// LS Electric XG5000 project: JG FRT C_MBR MAIN WELD
// PLC NewPLC
// module base 0 slot 0: 입력 모듈:XGI-D24A/B (DC 24V 입력, 32점 (전류소스 싱크공용/ 전류소스 입력))
// module base 0 slot 1: 출력 모듈:XGQ-TR4A/B (트랜지스터 출력, 32점 (0.1A용, 싱크출력/소스출력))
// module base 0 slot 2: 출력 모듈:XGQ-TR4A/B (트랜지스터 출력, 32점 (0.1A용, 싱크출력/소스출력))
// module base 0 slot 3: Rnet:XGL-RMEA/B (Rnet 통신 모듈, Rnet Master)
// module base 0 slot 4: Rnet:XGL-RMEA/B (Rnet 통신 모듈, Rnet Master)
// module base 0 slot 5: Rnet:XGL-RMEA/B (Rnet 통신 모듈, Rnet Master)
// module base 0 slot 6: Dnet:XGL-DMEA/B (Dnet 통신 모듈, DeviceNet Master)
// module base 0 slot 7: Dnet:XGL-DMEA/B (Dnet 통신 모듈, DeviceNet Master)
// module base 0 slot 8: FEnet:XGL-EFMT(B) (Fast Ethernet 통신 모듈, 전기 Master)
// module base 0 slot 9: FEnet:XGL-EFMT(B) (Fast Ethernet 통신 모듈, 전기 Master)

PROGRAM Main (task: 스캔 프로그램)

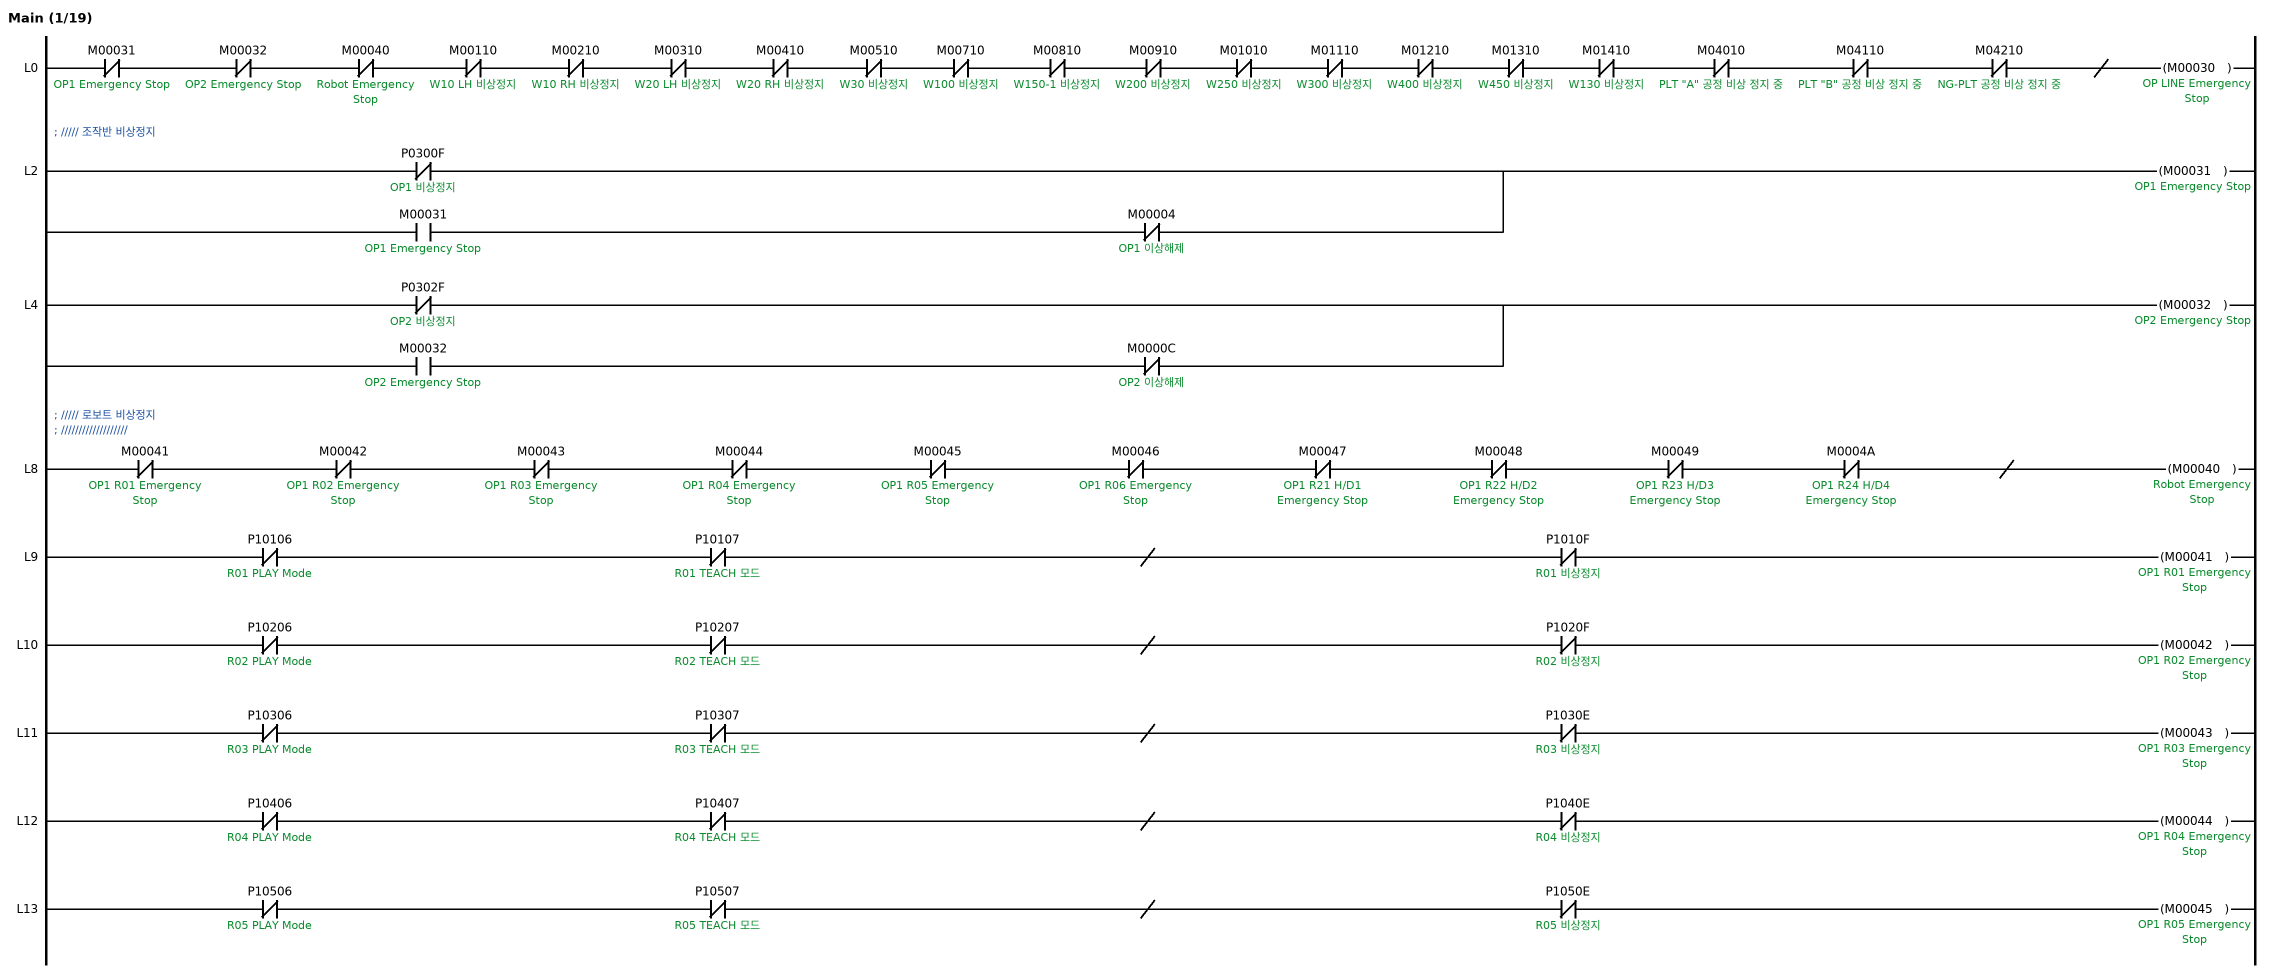
; L0
LOAD NOT  M00031	// OP1 Emergency Stop
AND NOT   M00032	// OP2 Emergency Stop
AND NOT   M00040	// Robot Emergency Stop
AND NOT   M00110	// W10 LH 비상정지
AND NOT   M00210	// W10 RH 비상정지
AND NOT   M00310	// W20 LH 비상정지
AND NOT   M00410	// W20 RH 비상정지
AND NOT   M00510	// W30 비상정지
AND NOT   M00710	// W100 비상정지
AND NOT   M00810	// W150-1 비상정지
AND NOT   M00910	// W200 비상정지
AND NOT   M01010	// W250 비상정지
AND NOT   M01110	// W300 비상정지
AND NOT   M01210	// W400 비상정지
AND NOT   M01310	// W450 비상정지
AND NOT   M01410	// W130 비상정지
AND NOT   M04010	// PLT "A" 공정 비상 정지 중
AND NOT   M04110	// PLT "B" 공정 비상 정지 중
AND NOT   M04210	// NG-PLT 공정 비상 정지 중
NOT
OUT       M00030	// OP LINE Emergency Stop
// ///// 조작반 비상정지
; L2
LOAD NOT  P0300F	// OP1 비상정지
LOAD      M00031	// OP1 Emergency Stop
AND NOT   M00004	// OP1 이상해제
OR LOAD
OUT       M00031	// OP1 Emergency Stop
; L4
LOAD NOT  P0302F	// OP2 비상정지
LOAD      M00032	// OP2 Emergency Stop
AND NOT   M0000C	// OP2 이상해제
OR LOAD
OUT       M00032	// OP2 Emergency Stop
// ///// 로보트 비상정지
// ///////////////////
; L8
LOAD NOT  M00041	// OP1 R01 Emergency Stop
AND NOT   M00042	// OP1 R02 Emergency Stop
AND NOT   M00043	// OP1 R03 Emergency Stop
AND NOT   M00044	// OP1 R04 Emergency Stop
AND NOT   M00045	// OP1 R05 Emergency Stop
AND NOT   M00046	// OP1 R06 Emergency Stop
AND NOT   M00047	// OP1 R21 H/D1 Emergency Stop
AND NOT   M00048	// OP1 R22 H/D2 Emergency Stop
AND NOT   M00049	// OP1 R23 H/D3 Emergency Stop
AND NOT   M0004A	// OP1 R24 H/D4 Emergency Stop
NOT
OUT       M00040	// Robot Emergency Stop
; L9
LOAD NOT  P10106	// R01 PLAY Mode
AND NOT   P10107	// R01 TEACH 모드
NOT
AND NOT   P1010F	// R01 비상정지
OUT       M00041	// OP1 R01 Emergency Stop
; L10
LOAD NOT  P10206	// R02 PLAY Mode
AND NOT   P10207	// R02 TEACH 모드
NOT
AND NOT   P1020F	// R02 비상정지
OUT       M00042	// OP1 R02 Emergency Stop
; L11
LOAD NOT  P10306	// R03 PLAY Mode
AND NOT   P10307	// R03 TEACH 모드
NOT
AND NOT   P1030E	// R03 비상정지
OUT       M00043	// OP1 R03 Emergency Stop
; L12
LOAD NOT  P10406	// R04 PLAY Mode
AND NOT   P10407	// R04 TEACH 모드
NOT
AND NOT   P1040E	// R04 비상정지
OUT       M00044	// OP1 R04 Emergency Stop
; L13
LOAD NOT  P10506	// R05 PLAY Mode
AND NOT   P10507	// R05 TEACH 모드
NOT
AND NOT   P1050E	// R05 비상정지
OUT       M00045	// OP1 R05 Emergency Stop

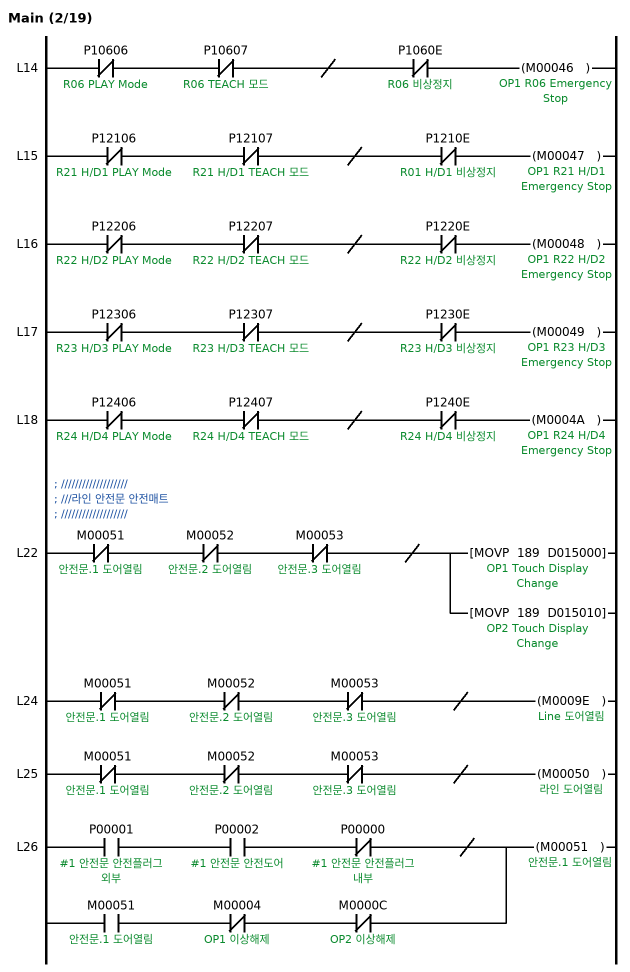
; L14
LOAD NOT  P10606	// R06 PLAY Mode
AND NOT   P10607	// R06 TEACH 모드
NOT
AND NOT   P1060E	// R06 비상정지
OUT       M00046	// OP1 R06 Emergency Stop
; L15
LOAD NOT  P12106	// R21 H/D1 PLAY Mode
AND NOT   P12107	// R21 H/D1 TEACH 모드
NOT
AND NOT   P1210E	// R01 H/D1 비상정지
OUT       M00047	// OP1 R21 H/D1 Emergency Stop
; L16
LOAD NOT  P12206	// R22 H/D2 PLAY Mode
AND NOT   P12207	// R22 H/D2 TEACH 모드
NOT
AND NOT   P1220E	// R22 H/D2 비상정지
OUT       M00048	// OP1 R22 H/D2 Emergency Stop
; L17
LOAD NOT  P12306	// R23 H/D3 PLAY Mode
AND NOT   P12307	// R23 H/D3 TEACH 모드
NOT
AND NOT   P1230E	// R23 H/D3 비상정지
OUT       M00049	// OP1 R23 H/D3 Emergency Stop
; L18
LOAD NOT  P12406	// R24 H/D4 PLAY Mode
AND NOT   P12407	// R24 H/D4 TEACH 모드
NOT
AND NOT   P1240E	// R24 H/D4 비상정지
OUT       M0004A	// OP1 R24 H/D4 Emergency Stop
// ///////////////////
// ///라인 안전문 안전매트
// ///////////////////
; L22
LOAD NOT  M00051	// 안전문.1 도어열림
AND NOT   M00052	// 안전문.2 도어열림
AND NOT   M00053	// 안전문.3 도어열림
NOT
MOVP      189 D015000	// OP1 Touch Display Change
MOVP      189 D015010	// OP2 Touch Display Change
; L24
LOAD NOT  M00051	// 안전문.1 도어열림
AND NOT   M00052	// 안전문.2 도어열림
AND NOT   M00053	// 안전문.3 도어열림
NOT
OUT       M0009E	// Line 도어열림
; L25
LOAD NOT  M00051	// 안전문.1 도어열림
AND NOT   M00052	// 안전문.2 도어열림
AND NOT   M00053	// 안전문.3 도어열림
NOT
OUT       M00050	// 라인 도어열림
; L26
LOAD      P00001	// #1 안전문 안전플러그 외부
AND       P00002	// #1 안전문 안전도어
AND NOT   P00000	// #1 안전문 안전플러그 내부
NOT
LOAD      M00051	// 안전문.1 도어열림
AND NOT   M00004	// OP1 이상해제
AND NOT   M0000C	// OP2 이상해제
OR LOAD
OUT       M00051	// 안전문.1 도어열림

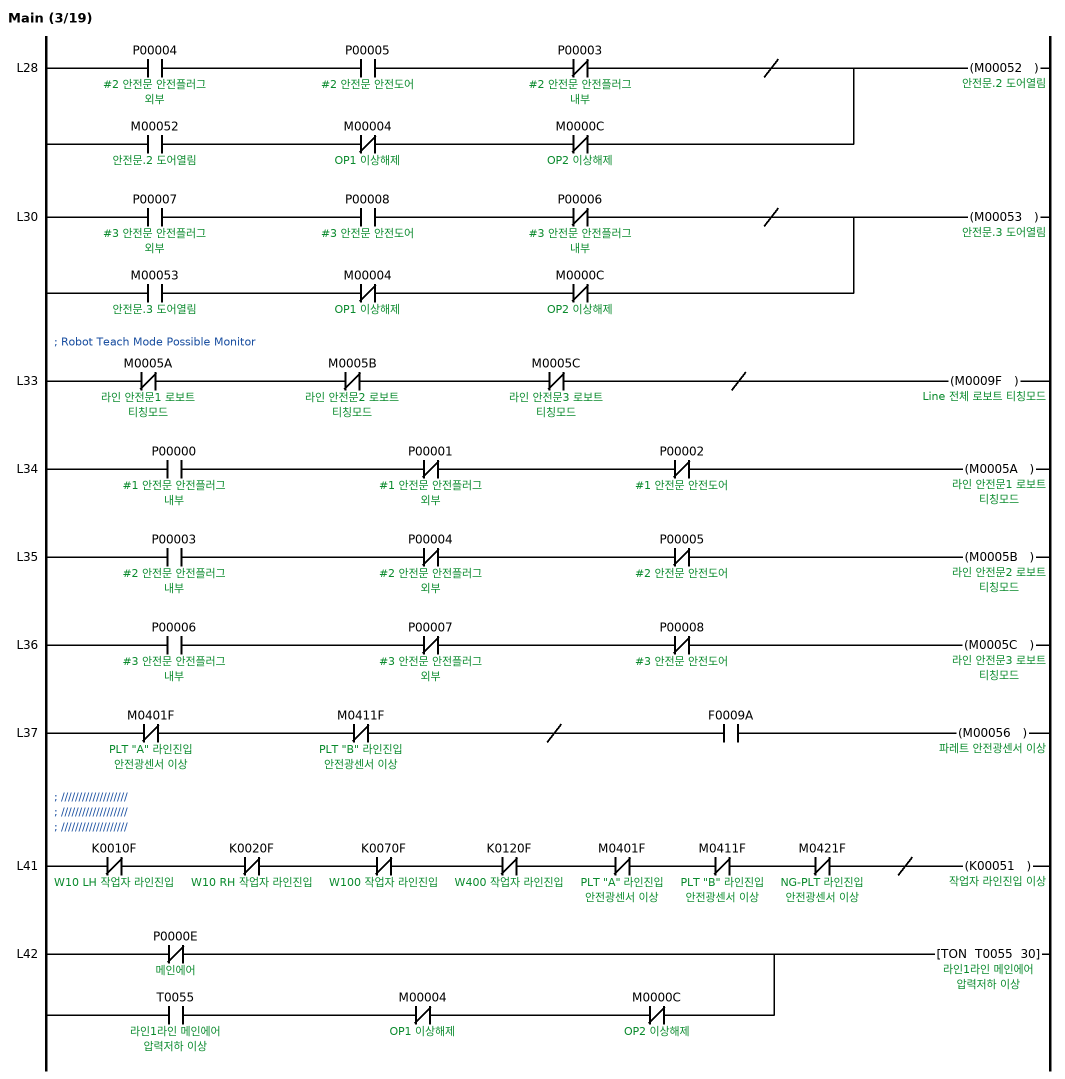
; L28
LOAD      P00004	// #2 안전문 안전플러그 외부
AND       P00005	// #2 안전문 안전도어
AND NOT   P00003	// #2 안전문 안전플러그 내부
NOT
LOAD      M00052	// 안전문.2 도어열림
AND NOT   M00004	// OP1 이상해제
AND NOT   M0000C	// OP2 이상해제
OR LOAD
OUT       M00052	// 안전문.2 도어열림
; L30
LOAD      P00007	// #3 안전문 안전플러그 외부
AND       P00008	// #3 안전문 안전도어
AND NOT   P00006	// #3 안전문 안전플러그 내부
NOT
LOAD      M00053	// 안전문.3 도어열림
AND NOT   M00004	// OP1 이상해제
AND NOT   M0000C	// OP2 이상해제
OR LOAD
OUT       M00053	// 안전문.3 도어열림
// Robot Teach Mode Possible Monitor
; L33
LOAD NOT  M0005A	// 라인 안전문1 로보트 티칭모드
AND NOT   M0005B	// 라인 안전문2 로보트 티칭모드
AND NOT   M0005C	// 라인 안전문3 로보트 티칭모드
NOT
OUT       M0009F	// Line 전체 로보트 티칭모드
; L34
LOAD      P00000	// #1 안전문 안전플러그 내부
AND NOT   P00001	// #1 안전문 안전플러그 외부
AND NOT   P00002	// #1 안전문 안전도어
OUT       M0005A	// 라인 안전문1 로보트 티칭모드
; L35
LOAD      P00003	// #2 안전문 안전플러그 내부
AND NOT   P00004	// #2 안전문 안전플러그 외부
AND NOT   P00005	// #2 안전문 안전도어
OUT       M0005B	// 라인 안전문2 로보트 티칭모드
; L36
LOAD      P00006	// #3 안전문 안전플러그 내부
AND NOT   P00007	// #3 안전문 안전플러그 외부
AND NOT   P00008	// #3 안전문 안전도어
OUT       M0005C	// 라인 안전문3 로보트 티칭모드
; L37
LOAD NOT  M0401F	// PLT "A" 라인진입 안전광센서 이상
AND NOT   M0411F	// PLT "B" 라인진입 안전광센서 이상
NOT
AND       F0009A
OUT       M00056	// 파레트 안전광센서 이상
// ///////////////////
// ///////////////////
// ///////////////////
; L41
LOAD NOT  K0010F	// W10 LH 작업자 라인진입
AND NOT   K0020F	// W10 RH 작업자 라인진입
AND NOT   K0070F	// W100 작업자 라인진입
AND NOT   K0120F	// W400 작업자 라인진입
AND NOT   M0401F	// PLT "A" 라인진입 안전광센서 이상
AND NOT   M0411F	// PLT "B" 라인진입 안전광센서 이상
AND NOT   M0421F	// NG-PLT 라인진입 안전광센서 이상
NOT
OUT       K00051	//  작업자 라인진입 이상
; L42
LOAD NOT  P0000E	// 메인에어
LOAD      T0055	// 라인1라인 메인에어 압력저하 이상
AND NOT   M00004	// OP1 이상해제
AND NOT   M0000C	// OP2 이상해제
OR LOAD
TON       T0055 30	// 라인1라인 메인에어 압력저하 이상

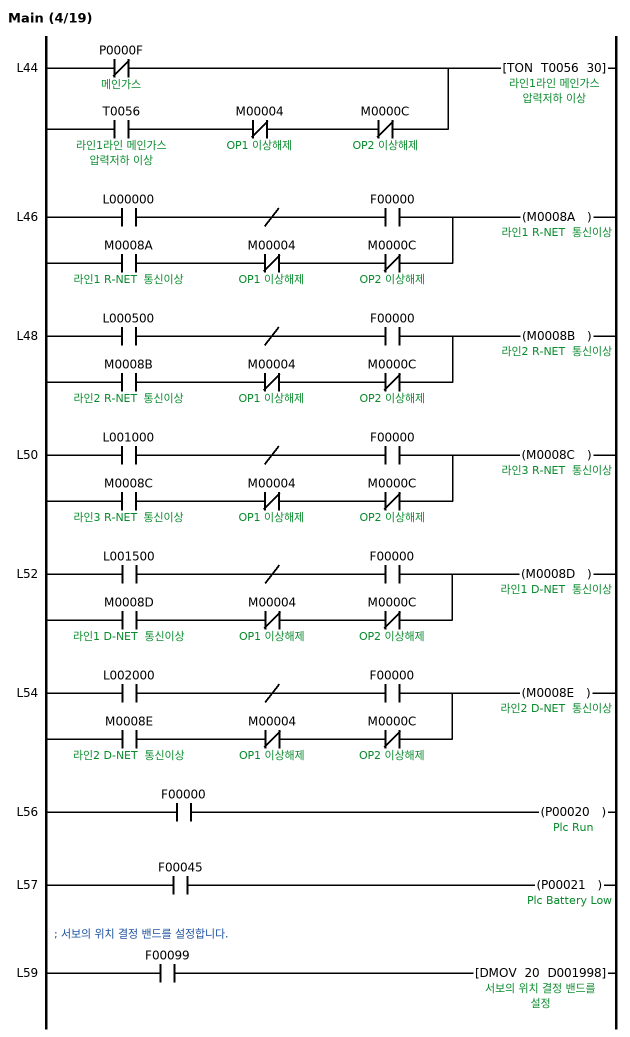
; L44
LOAD NOT  P0000F	// 메인가스
LOAD      T0056	// 라인1라인 메인가스 압력저하 이상
AND NOT   M00004	// OP1 이상해제
AND NOT   M0000C	// OP2 이상해제
OR LOAD
TON       T0056 30	// 라인1라인 메인가스 압력저하 이상
; L46
LOAD      L000000
NOT
AND       F00000
LOAD      M0008A	// 라인1 R-NET  통신이상
AND NOT   M00004	// OP1 이상해제
AND NOT   M0000C	// OP2 이상해제
OR LOAD
OUT       M0008A	// 라인1 R-NET  통신이상
; L48
LOAD      L000500
NOT
AND       F00000
LOAD      M0008B	// 라인2 R-NET  통신이상
AND NOT   M00004	// OP1 이상해제
AND NOT   M0000C	// OP2 이상해제
OR LOAD
OUT       M0008B	// 라인2 R-NET  통신이상
; L50
LOAD      L001000
NOT
AND       F00000
LOAD      M0008C	// 라인3 R-NET  통신이상
AND NOT   M00004	// OP1 이상해제
AND NOT   M0000C	// OP2 이상해제
OR LOAD
OUT       M0008C	// 라인3 R-NET  통신이상
; L52
LOAD      L001500
NOT
AND       F00000
LOAD      M0008D	// 라인1 D-NET  통신이상
AND NOT   M00004	// OP1 이상해제
AND NOT   M0000C	// OP2 이상해제
OR LOAD
OUT       M0008D	// 라인1 D-NET  통신이상
; L54
LOAD      L002000
NOT
AND       F00000
LOAD      M0008E	// 라인2 D-NET  통신이상
AND NOT   M00004	// OP1 이상해제
AND NOT   M0000C	// OP2 이상해제
OR LOAD
OUT       M0008E	// 라인2 D-NET  통신이상
; L56
LOAD      F00000
OUT       P00020	// Plc Run
; L57
LOAD      F00045
OUT       P00021	// Plc Battery Low
// 서보의 위치 결정 밴드를 설정합니다.
; L59
LOAD      F00099
DMOV      20 D001998	// 서보의 위치 결정 밴드를 설정

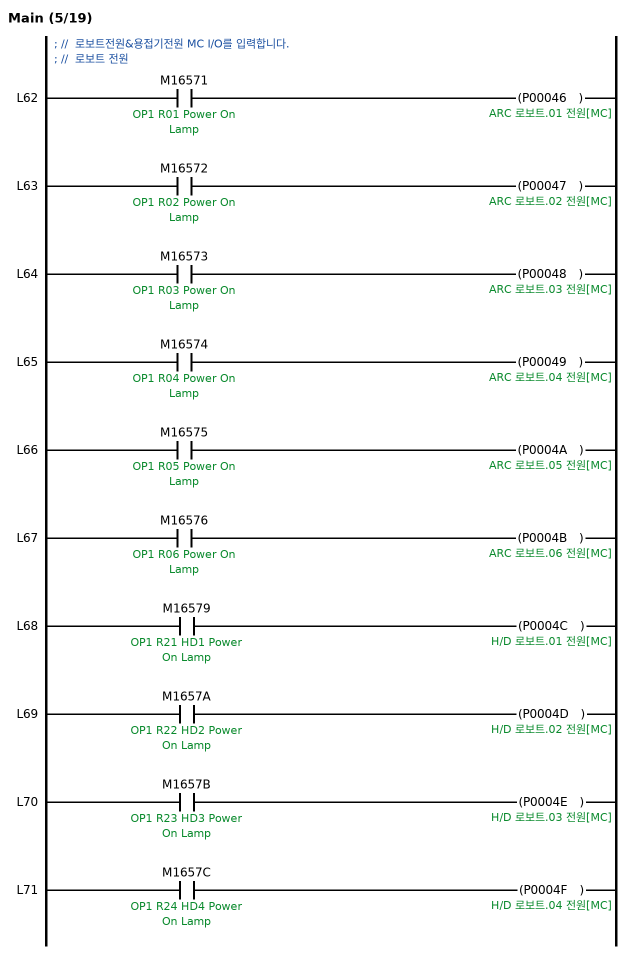
//   //  로보트전원&용접기전원 MC I/O를 입력합니다.
//   //  로보트 전원
; L62
LOAD      M16571	// OP1 R01 Power On Lamp
OUT       P00046	// ARC 로보트.01 전원[MC]
; L63
LOAD      M16572	// OP1 R02 Power On Lamp
OUT       P00047	// ARC 로보트.02 전원[MC]
; L64
LOAD      M16573	// OP1 R03 Power On Lamp
OUT       P00048	// ARC 로보트.03 전원[MC]
; L65
LOAD      M16574	// OP1 R04 Power On Lamp
OUT       P00049	// ARC 로보트.04 전원[MC]
; L66
LOAD      M16575	// OP1 R05 Power On Lamp
OUT       P0004A	// ARC 로보트.05 전원[MC]
; L67
LOAD      M16576	// OP1 R06 Power On Lamp
OUT       P0004B	// ARC 로보트.06 전원[MC]
; L68
LOAD      M16579	// OP1 R21 HD1 Power On Lamp
OUT       P0004C	// H/D 로보트.01 전원[MC]
; L69
LOAD      M1657A	// OP1 R22 HD2 Power On Lamp
OUT       P0004D	// H/D 로보트.02 전원[MC]
; L70
LOAD      M1657B	// OP1 R23 HD3 Power On Lamp
OUT       P0004E	// H/D 로보트.03 전원[MC]
; L71
LOAD      M1657C	// OP1 R24 HD4 Power On Lamp
OUT       P0004F	// H/D 로보트.04 전원[MC]

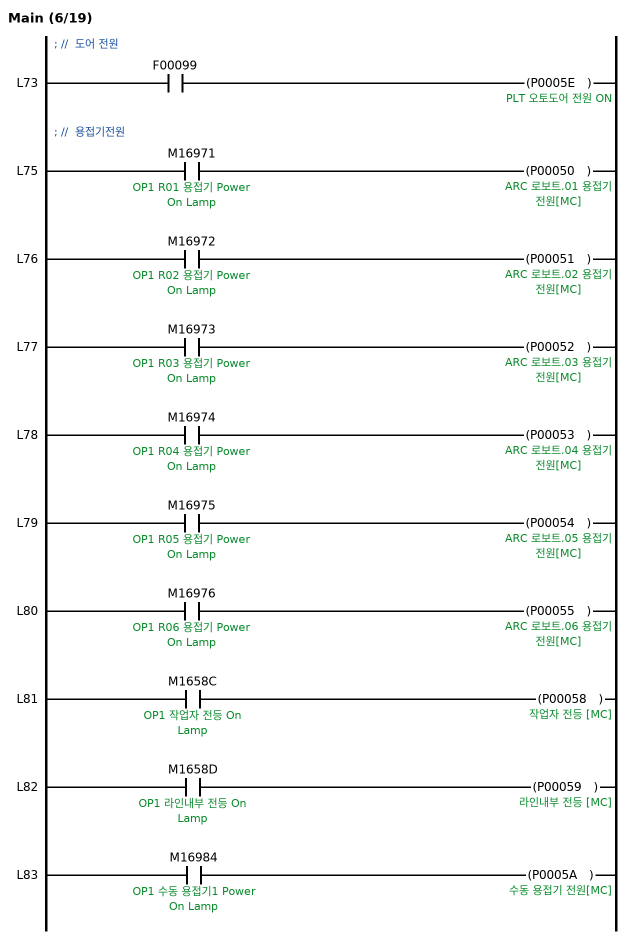
//   //  도어 전원
; L73
LOAD      F00099
OUT       P0005E	// PLT 오토도어 전원 ON
//   //  용접기전원
; L75
LOAD      M16971	// OP1 R01 용접기 Power On Lamp
OUT       P00050	// ARC 로보트.01 용접기 전원[MC]
; L76
LOAD      M16972	// OP1 R02 용접기 Power On Lamp
OUT       P00051	// ARC 로보트.02 용접기 전원[MC]
; L77
LOAD      M16973	// OP1 R03 용접기 Power On Lamp
OUT       P00052	// ARC 로보트.03 용접기 전원[MC]
; L78
LOAD      M16974	// OP1 R04 용접기 Power On Lamp
OUT       P00053	// ARC 로보트.04 용접기 전원[MC]
; L79
LOAD      M16975	// OP1 R05 용접기 Power On Lamp
OUT       P00054	// ARC 로보트.05 용접기 전원[MC]
; L80
LOAD      M16976	// OP1 R06 용접기 Power On Lamp
OUT       P00055	// ARC 로보트.06 용접기 전원[MC]
; L81
LOAD      M1658C	// OP1 작업자 전등 On Lamp
OUT       P00058	// 작업자 전등 [MC]
; L82
LOAD      M1658D	// OP1 라인내부 전등 On Lamp
OUT       P00059	// 라인내부 전등 [MC]
; L83
LOAD      M16984	// OP1 수동 용접기1 Power On Lamp
OUT       P0005A	// 수동 용접기 전원[MC]

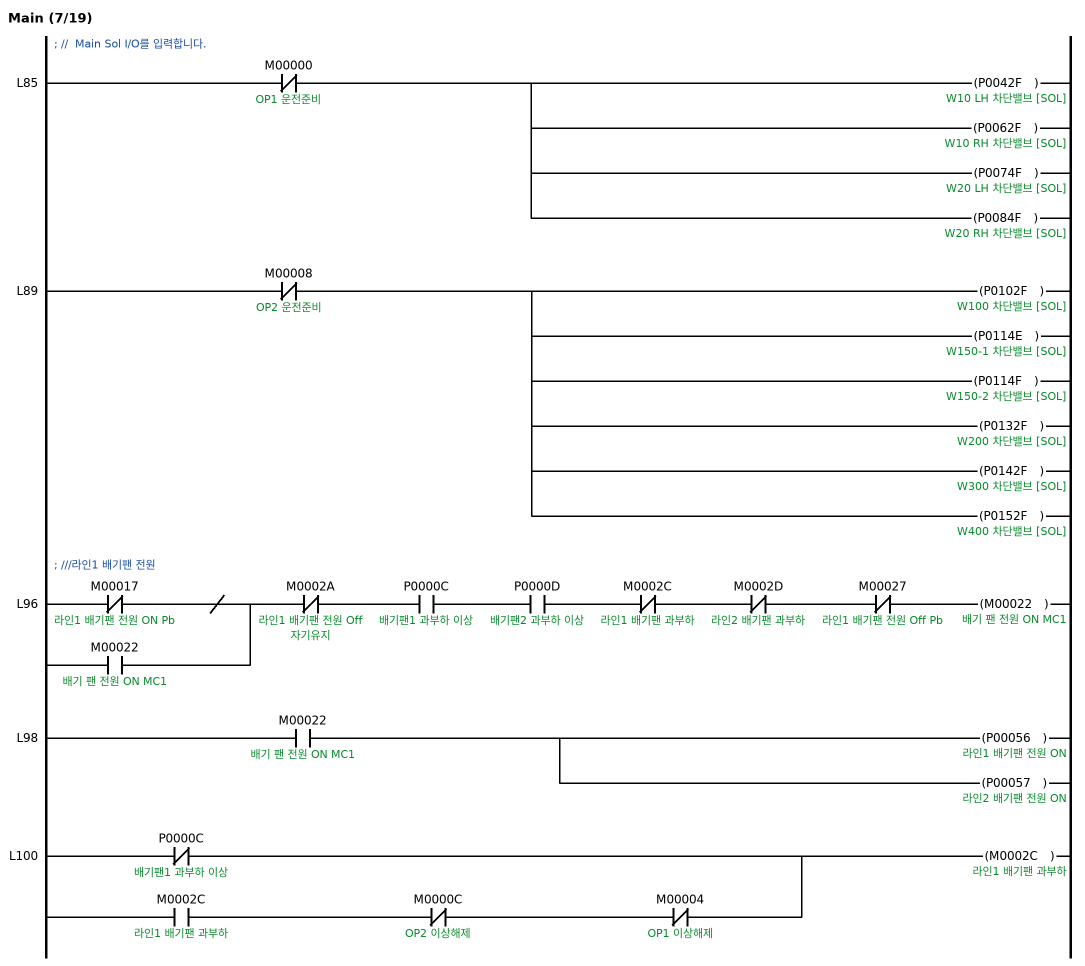
//   //  Main Sol I/O를 입력합니다.
; L85
LOAD NOT  M00000	// OP1 운전준비
OUT       P0042F	// W10 LH 차단밸브 [SOL]
OUT       P0062F	// W10 RH 차단밸브 [SOL]
OUT       P0074F	// W20 LH 차단밸브 [SOL]
OUT       P0084F	// W20 RH 차단밸브 [SOL]
; L89
LOAD NOT  M00008	// OP2 운전준비
OUT       P0102F	// W100 차단밸브 [SOL]
OUT       P0114E	// W150-1 차단밸브 [SOL]
OUT       P0114F	// W150-2 차단밸브 [SOL]
OUT       P0132F	// W200 차단밸브 [SOL]
OUT       P0142F	// W300 차단밸브 [SOL]
OUT       P0152F	// W400 차단밸브 [SOL]
// ///라인1 배기팬 전원
; L96
LOAD NOT  M00017	// 라인1 배기팬 전원 ON Pb
NOT
OR        M00022	// 배기 팬 전원 ON MC1
AND NOT   M0002A	// 라인1 배기팬 전원 Off 자기유지
AND       P0000C	// 배기팬1 과부하 이상
AND       P0000D	// 배기팬2 과부하 이상
AND NOT   M0002C	// 라인1 배기팬 과부하
AND NOT   M0002D	// 라인2 배기팬 과부하
AND NOT   M00027	// 라인1 배기팬 전원 Off Pb
OUT       M00022	// 배기 팬 전원 ON MC1
; L98
LOAD      M00022	// 배기 팬 전원 ON MC1
OUT       P00056	// 라인1 배기팬 전원 ON
OUT       P00057	// 라인2 배기팬 전원 ON
; L100
LOAD NOT  P0000C	// 배기팬1 과부하 이상
LOAD      M0002C	// 라인1 배기팬 과부하
AND NOT   M0000C	// OP2 이상해제
AND NOT   M00004	// OP1 이상해제
OR LOAD
OUT       M0002C	// 라인1 배기팬 과부하

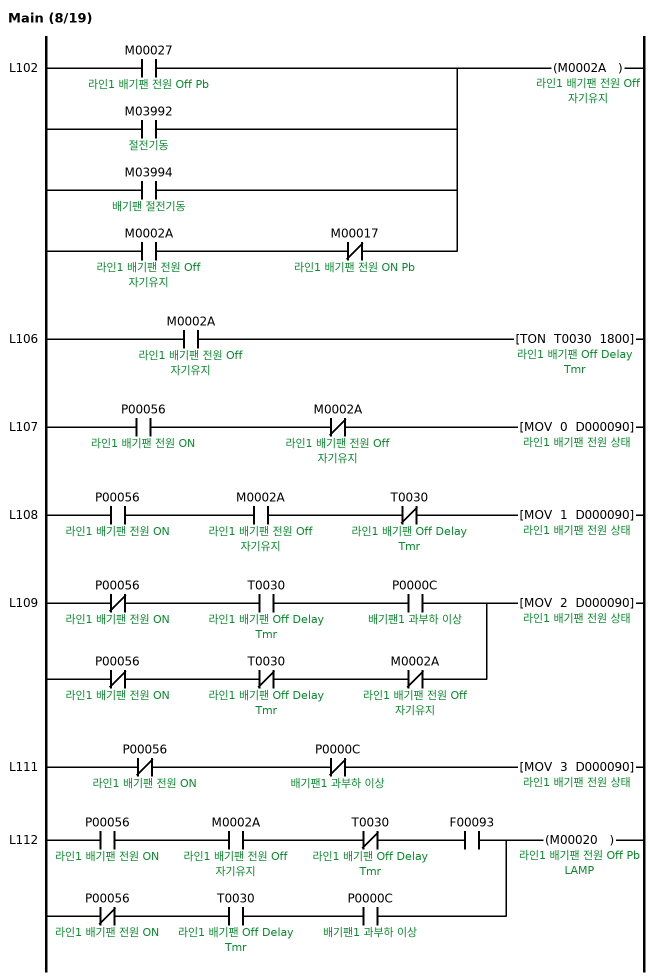
; L102
LOAD      M00027	// 라인1 배기팬 전원 Off Pb
OR        M03992	// 절전기동
OR        M03994	// 배기팬 절전기동
LOAD      M0002A	// 라인1 배기팬 전원 Off 자기유지
AND NOT   M00017	// 라인1 배기팬 전원 ON Pb
OR LOAD
OUT       M0002A	// 라인1 배기팬 전원 Off 자기유지
; L106
LOAD      M0002A	// 라인1 배기팬 전원 Off 자기유지
TON       T0030 1800	// 라인1 배기팬 Off Delay Tmr
; L107
LOAD      P00056	// 라인1 배기팬 전원 ON
AND NOT   M0002A	// 라인1 배기팬 전원 Off 자기유지
MOV       0 D000090	// 라인1 배기팬 전원 상태
; L108
LOAD      P00056	// 라인1 배기팬 전원 ON
AND       M0002A	// 라인1 배기팬 전원 Off 자기유지
AND NOT   T0030	// 라인1 배기팬 Off Delay Tmr
MOV       1 D000090	// 라인1 배기팬 전원 상태
; L109
LOAD NOT  P00056	// 라인1 배기팬 전원 ON
AND       T0030	// 라인1 배기팬 Off Delay Tmr
AND       P0000C	// 배기팬1 과부하 이상
LOAD NOT  P00056	// 라인1 배기팬 전원 ON
AND NOT   T0030	// 라인1 배기팬 Off Delay Tmr
AND NOT   M0002A	// 라인1 배기팬 전원 Off 자기유지
OR LOAD
MOV       2 D000090	// 라인1 배기팬 전원 상태
; L111
LOAD NOT  P00056	// 라인1 배기팬 전원 ON
AND NOT   P0000C	// 배기팬1 과부하 이상
MOV       3 D000090	// 라인1 배기팬 전원 상태
; L112
LOAD      P00056	// 라인1 배기팬 전원 ON
AND       M0002A	// 라인1 배기팬 전원 Off 자기유지
AND NOT   T0030	// 라인1 배기팬 Off Delay Tmr
AND       F00093
LOAD NOT  P00056	// 라인1 배기팬 전원 ON
AND       T0030	// 라인1 배기팬 Off Delay Tmr
AND       P0000C	// 배기팬1 과부하 이상
OR LOAD
OUT       M00020	// 라인1 배기팬 전원 Off Pb LAMP

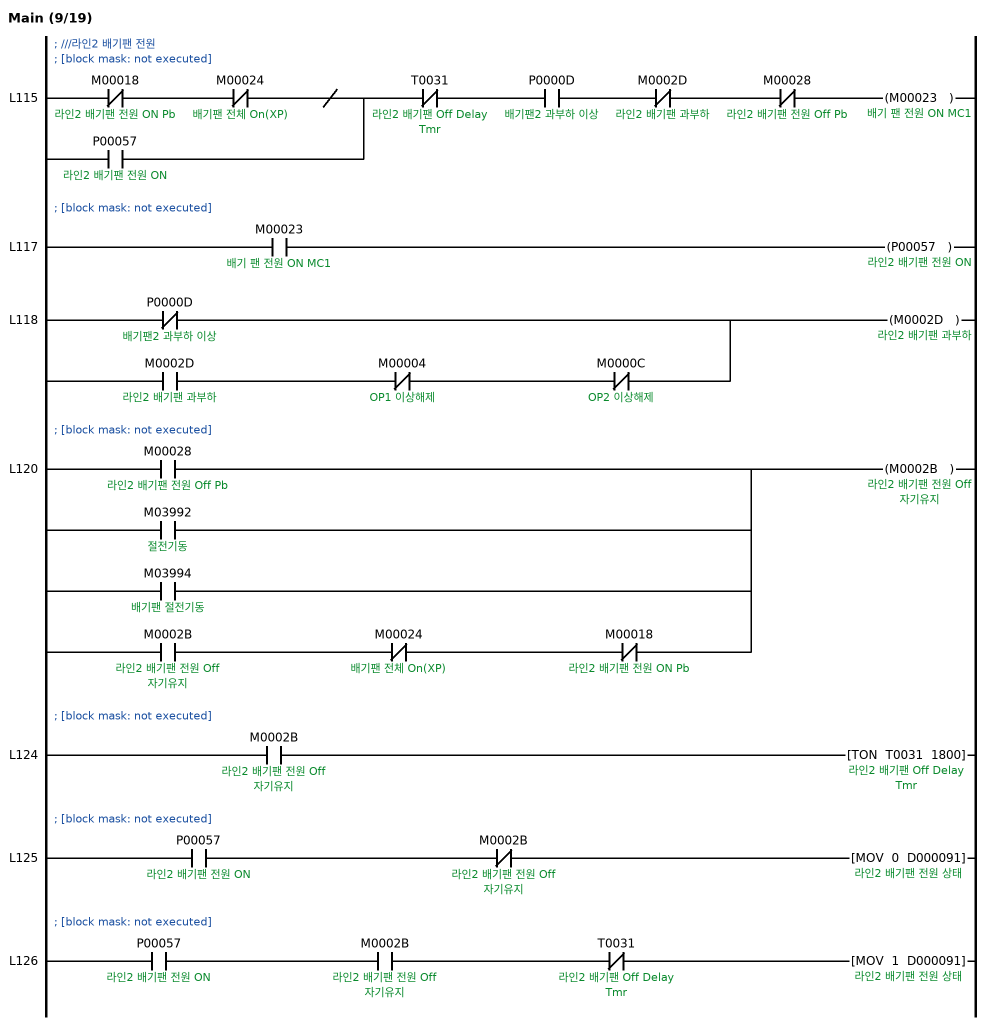
// ///라인2 배기팬 전원
; L115 (block mask: not executed)
LOAD NOT  M00018	// 라인2 배기팬 전원 ON Pb
AND NOT   M00024	// 배기팬 전체 On(XP)
NOT
OR        P00057	// 라인2 배기팬 전원 ON
AND NOT   T0031	// 라인2 배기팬 Off Delay Tmr
AND       P0000D	// 배기팬2 과부하 이상
AND NOT   M0002D	// 라인2 배기팬 과부하
AND NOT   M00028	// 라인2 배기팬 전원 Off Pb
OUT       M00023	// 배기 팬 전원 ON MC1
; L117 (block mask: not executed)
LOAD      M00023	// 배기 팬 전원 ON MC1
OUT       P00057	// 라인2 배기팬 전원 ON
; L118
LOAD NOT  P0000D	// 배기팬2 과부하 이상
LOAD      M0002D	// 라인2 배기팬 과부하
AND NOT   M00004	// OP1 이상해제
AND NOT   M0000C	// OP2 이상해제
OR LOAD
OUT       M0002D	// 라인2 배기팬 과부하
; L120 (block mask: not executed)
LOAD      M00028	// 라인2 배기팬 전원 Off Pb
OR        M03992	// 절전기동
OR        M03994	// 배기팬 절전기동
LOAD      M0002B	// 라인2 배기팬 전원 Off 자기유지
AND NOT   M00024	// 배기팬 전체 On(XP)
AND NOT   M00018	// 라인2 배기팬 전원 ON Pb
OR LOAD
OUT       M0002B	// 라인2 배기팬 전원 Off 자기유지
; L124 (block mask: not executed)
LOAD      M0002B	// 라인2 배기팬 전원 Off 자기유지
TON       T0031 1800	// 라인2 배기팬 Off Delay Tmr
; L125 (block mask: not executed)
LOAD      P00057	// 라인2 배기팬 전원 ON
AND NOT   M0002B	// 라인2 배기팬 전원 Off 자기유지
MOV       0 D000091	// 라인2 배기팬 전원 상태
; L126 (block mask: not executed)
LOAD      P00057	// 라인2 배기팬 전원 ON
AND       M0002B	// 라인2 배기팬 전원 Off 자기유지
AND NOT   T0031	// 라인2 배기팬 Off Delay Tmr
MOV       1 D000091	// 라인2 배기팬 전원 상태

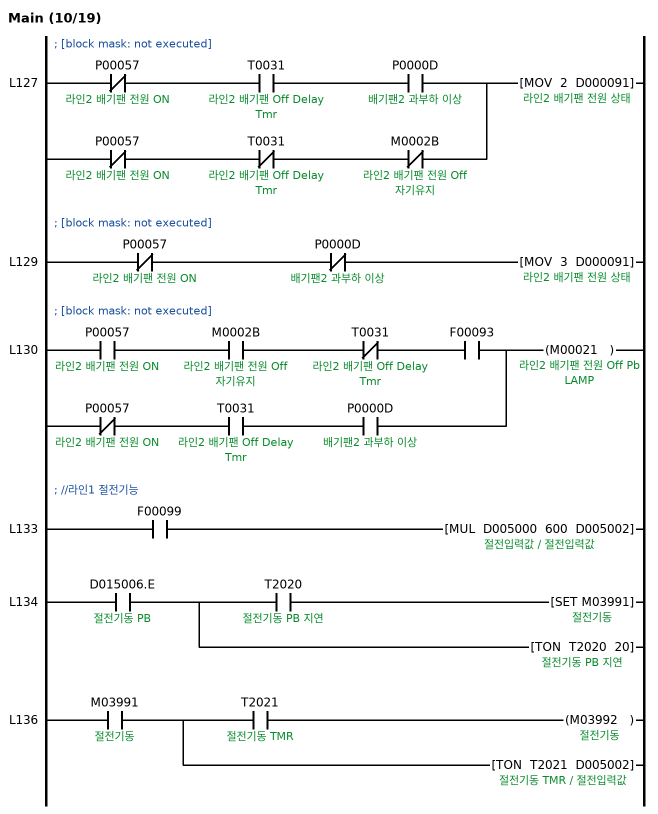
; L127 (block mask: not executed)
LOAD NOT  P00057	// 라인2 배기팬 전원 ON
AND       T0031	// 라인2 배기팬 Off Delay Tmr
AND       P0000D	// 배기팬2 과부하 이상
LOAD NOT  P00057	// 라인2 배기팬 전원 ON
AND NOT   T0031	// 라인2 배기팬 Off Delay Tmr
AND NOT   M0002B	// 라인2 배기팬 전원 Off 자기유지
OR LOAD
MOV       2 D000091	// 라인2 배기팬 전원 상태
; L129 (block mask: not executed)
LOAD NOT  P00057	// 라인2 배기팬 전원 ON
AND NOT   P0000D	// 배기팬2 과부하 이상
MOV       3 D000091	// 라인2 배기팬 전원 상태
; L130 (block mask: not executed)
LOAD      P00057	// 라인2 배기팬 전원 ON
AND       M0002B	// 라인2 배기팬 전원 Off 자기유지
AND NOT   T0031	// 라인2 배기팬 Off Delay Tmr
AND       F00093
LOAD NOT  P00057	// 라인2 배기팬 전원 ON
AND       T0031	// 라인2 배기팬 Off Delay Tmr
AND       P0000D	// 배기팬2 과부하 이상
OR LOAD
OUT       M00021	// 라인2 배기팬 전원 Off Pb LAMP
//  //라인1 절전기능
; L133
LOAD      F00099
MUL       D005000 600 D005002	// 절전입력값 / 절전입력값
; L134
LOAD      D015006.E	// 절전기동 PB
MPUSH
AND       T2020	// 절전기동 PB 지연
SET       M03991	// 절전기동
MPOP
TON       T2020 20	// 절전기동 PB 지연
; L136
LOAD      M03991	// 절전기동
MPUSH
AND       T2021	// 절전기동 TMR
OUT       M03992	// 절전기동
MPOP
TON       T2021 D005002	// 절전기동 TMR / 절전입력값

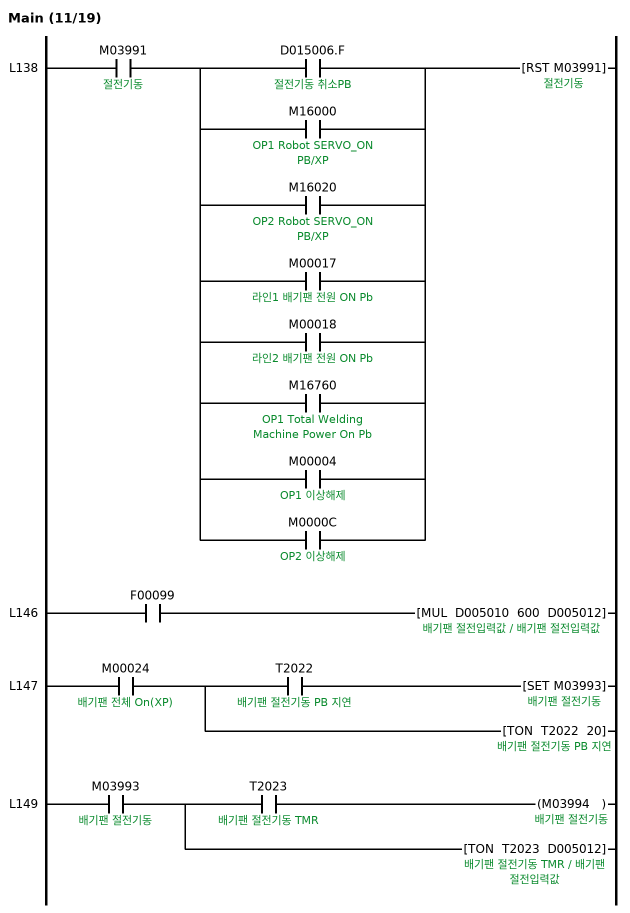
; L138
LOAD      M03991	// 절전기동
LOAD      D015006.F	// 절전기동 취소PB
OR        M16000	// OP1 Robot SERVO_ON PB/XP
OR        M16020	// OP2 Robot SERVO_ON PB/XP
OR        M00017	// 라인1 배기팬 전원 ON Pb
OR        M00018	// 라인2 배기팬 전원 ON Pb
OR        M16760	// OP1 Total Welding Machine Power On Pb
OR        M00004	// OP1 이상해제
OR        M0000C	// OP2 이상해제
AND LOAD
RST       M03991	// 절전기동
; L146
LOAD      F00099
MUL       D005010 600 D005012	// 배기팬 절전입력값 / 배기팬 절전입력값
; L147
LOAD      M00024	// 배기팬 전체 On(XP)
MPUSH
AND       T2022	// 배기팬 절전기동 PB 지연
SET       M03993	// 배기팬 절전기동
MPOP
TON       T2022 20	// 배기팬 절전기동 PB 지연
; L149
LOAD      M03993	// 배기팬 절전기동
MPUSH
AND       T2023	// 배기팬 절전기동 TMR
OUT       M03994	// 배기팬 절전기동
MPOP
TON       T2023 D005012	// 배기팬 절전기동 TMR / 배기팬 절전입력값

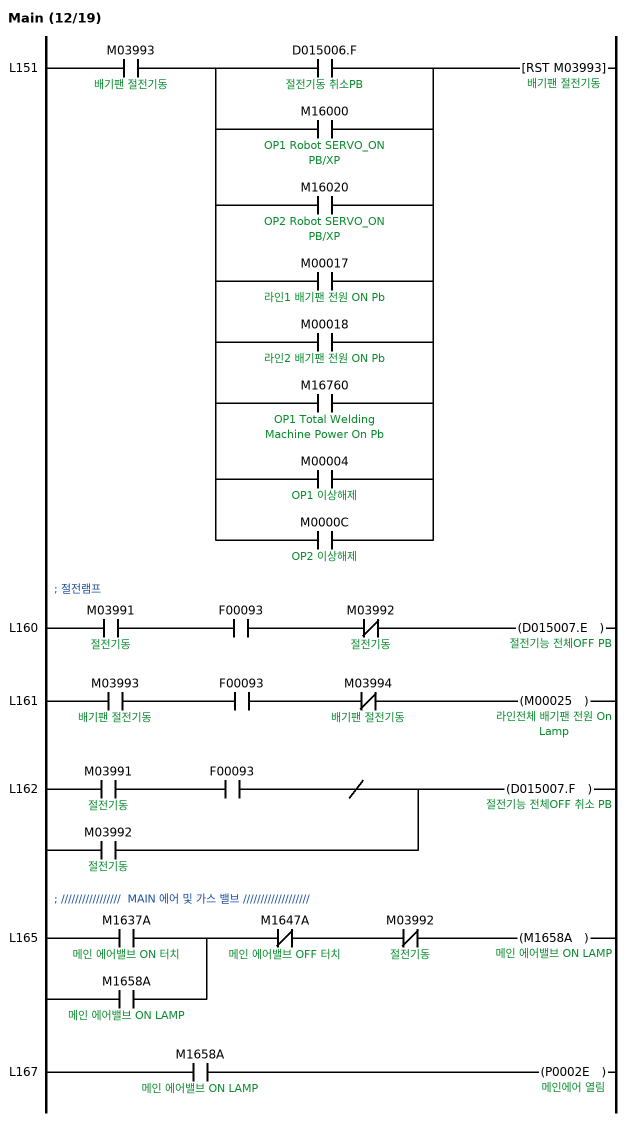
; L151
LOAD      M03993	// 배기팬 절전기동
LOAD      D015006.F	// 절전기동 취소PB
OR        M16000	// OP1 Robot SERVO_ON PB/XP
OR        M16020	// OP2 Robot SERVO_ON PB/XP
OR        M00017	// 라인1 배기팬 전원 ON Pb
OR        M00018	// 라인2 배기팬 전원 ON Pb
OR        M16760	// OP1 Total Welding Machine Power On Pb
OR        M00004	// OP1 이상해제
OR        M0000C	// OP2 이상해제
AND LOAD
RST       M03993	// 배기팬 절전기동
// 절전램프
; L160
LOAD      M03991	// 절전기동
AND       F00093
AND NOT   M03992	// 절전기동
OUT       D015007.E	// 절전기능 전체OFF PB
; L161
LOAD      M03993	// 배기팬 절전기동
AND       F00093
AND NOT   M03994	// 배기팬 절전기동
OUT       M00025	// 라인전체 배기팬 전원 On Lamp
; L162
LOAD      M03991	// 절전기동
AND       F00093
NOT
OR        M03992	// 절전기동
OUT       D015007.F	// 절전기능 전체OFF 취소 PB
// /////////////////  MAIN 에어 및 가스 밸브 ///////////////////
; L165
LOAD      M1637A	// 메인 에어밸브 ON 터치
OR        M1658A	// 메인 에어밸브 ON LAMP
AND NOT   M1647A	// 메인 에어밸브 OFF 터치
AND NOT   M03992	// 절전기동
OUT       M1658A	// 메인 에어밸브 ON LAMP
; L167
LOAD      M1658A	// 메인 에어밸브 ON LAMP
OUT       P0002E	// 메인에어 열림

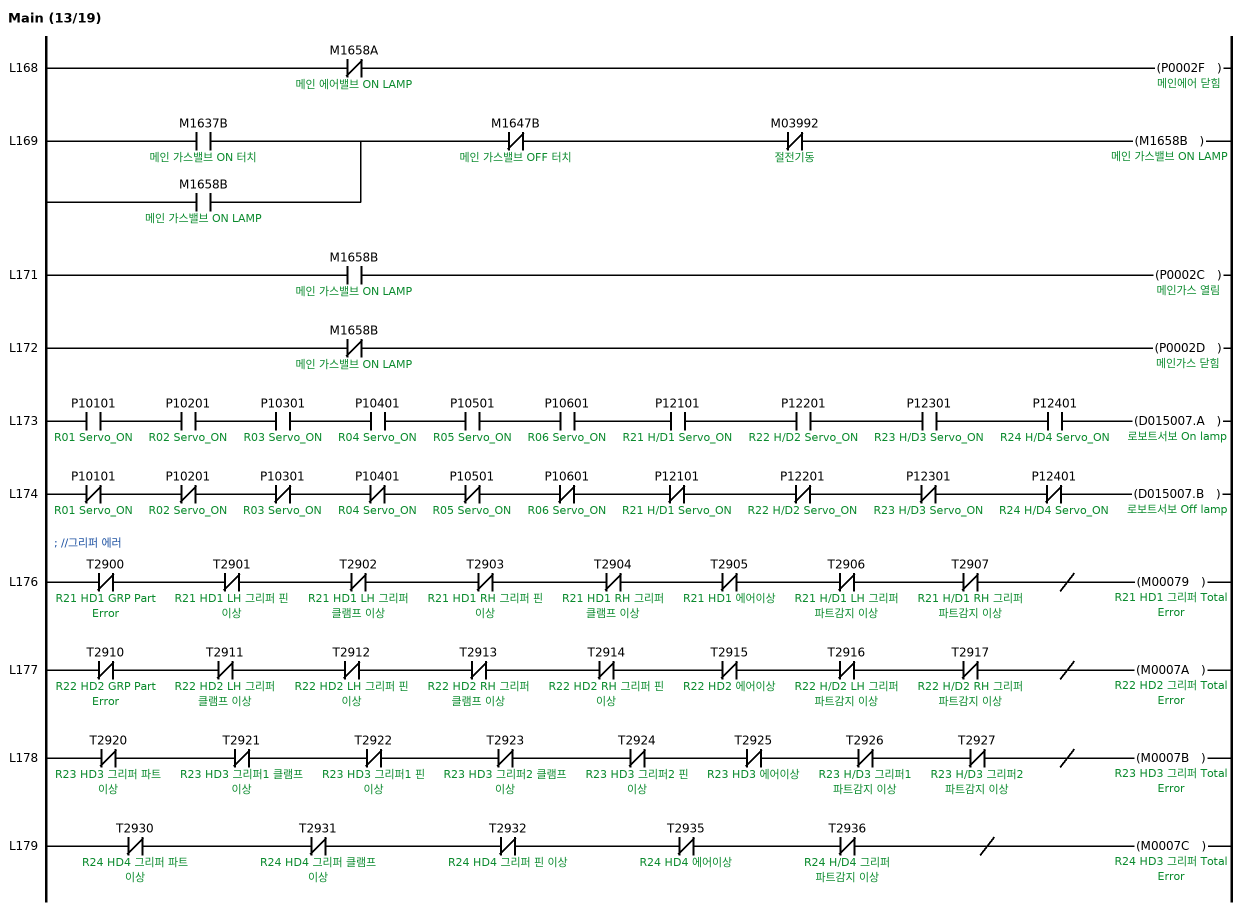
; L168
LOAD NOT  M1658A	// 메인 에어밸브 ON LAMP
OUT       P0002F	// 메인에어 닫힘
; L169
LOAD      M1637B	// 메인 가스밸브 ON 터치
OR        M1658B	// 메인 가스밸브 ON LAMP
AND NOT   M1647B	// 메인 가스밸브 OFF 터치
AND NOT   M03992	// 절전기동
OUT       M1658B	// 메인 가스밸브 ON LAMP
; L171
LOAD      M1658B	// 메인 가스밸브 ON LAMP
OUT       P0002C	// 메인가스 열림
; L172
LOAD NOT  M1658B	// 메인 가스밸브 ON LAMP
OUT       P0002D	// 메인가스 닫힘
; L173
LOAD      P10101	// R01 Servo_ON
AND       P10201	// R02 Servo_ON
AND       P10301	// R03 Servo_ON
AND       P10401	// R04 Servo_ON
AND       P10501	// R05 Servo_ON
AND       P10601	// R06 Servo_ON
AND       P12101	// R21 H/D1 Servo_ON
AND       P12201	// R22 H/D2 Servo_ON
AND       P12301	// R23 H/D3 Servo_ON
AND       P12401	// R24 H/D4 Servo_ON
OUT       D015007.A	// 로보트서보 On lamp
; L174
LOAD NOT  P10101	// R01 Servo_ON
AND NOT   P10201	// R02 Servo_ON
AND NOT   P10301	// R03 Servo_ON
AND NOT   P10401	// R04 Servo_ON
AND NOT   P10501	// R05 Servo_ON
AND NOT   P10601	// R06 Servo_ON
AND NOT   P12101	// R21 H/D1 Servo_ON
AND NOT   P12201	// R22 H/D2 Servo_ON
AND NOT   P12301	// R23 H/D3 Servo_ON
AND NOT   P12401	// R24 H/D4 Servo_ON
OUT       D015007.B	// 로보트서보 Off lamp
//  //그리퍼 에러
; L176
LOAD NOT  T2900	// R21 HD1 GRP Part Error 
AND NOT   T2901	// R21 HD1 LH 그리퍼 핀 이상
AND NOT   T2902	// R21 HD1 LH 그리퍼 클램프 이상
AND NOT   T2903	// R21 HD1 RH 그리퍼 핀 이상
AND NOT   T2904	// R21 HD1 RH 그리퍼 클램프 이상
AND NOT   T2905	// R21 HD1 에어이상
AND NOT   T2906	// R21 H/D1 LH 그리퍼 파트감지 이상
AND NOT   T2907	// R21 H/D1 RH 그리퍼 파트감지 이상
NOT
OUT       M00079	// R21 HD1 그리퍼 Total Error 
; L177
LOAD NOT  T2910	// R22 HD2 GRP Part Error 
AND NOT   T2911	// R22 HD2 LH 그리퍼 클램프 이상
AND NOT   T2912	// R22 HD2 LH 그리퍼 핀 이상
AND NOT   T2913	// R22 HD2 RH 그리퍼 클램프 이상
AND NOT   T2914	// R22 HD2 RH 그리퍼 핀 이상
AND NOT   T2915	// R22 HD2 에어이상
AND NOT   T2916	// R22 H/D2 LH 그리퍼 파트감지 이상
AND NOT   T2917	// R22 H/D2 RH 그리퍼 파트감지 이상
NOT
OUT       M0007A	// R22 HD2 그리퍼 Total Error 
; L178
LOAD NOT  T2920	// R23 HD3 그리퍼 파트 이상
AND NOT   T2921	// R23 HD3 그리퍼1 클램프 이상
AND NOT   T2922	// R23 HD3 그리퍼1 핀 이상
AND NOT   T2923	// R23 HD3 그리퍼2 클램프 이상
AND NOT   T2924	// R23 HD3 그리퍼2 핀 이상
AND NOT   T2925	// R23 HD3 에어이상
AND NOT   T2926	// R23 H/D3 그리퍼1 파트감지 이상
AND NOT   T2927	// R23 H/D3 그리퍼2 파트감지 이상
NOT
OUT       M0007B	// R23 HD3 그리퍼 Total Error 
; L179
LOAD NOT  T2930	// R24 HD4 그리퍼 파트 이상
AND NOT   T2931	// R24 HD4 그리퍼 클램프 이상
AND NOT   T2932	// R24 HD4 그리퍼 핀 이상
AND NOT   T2935	// R24 HD4 에어이상
AND NOT   T2936	// R24 H/D4 그리퍼 파트감지 이상
NOT
OUT       M0007C	// R24 HD3 그리퍼 Total Error 

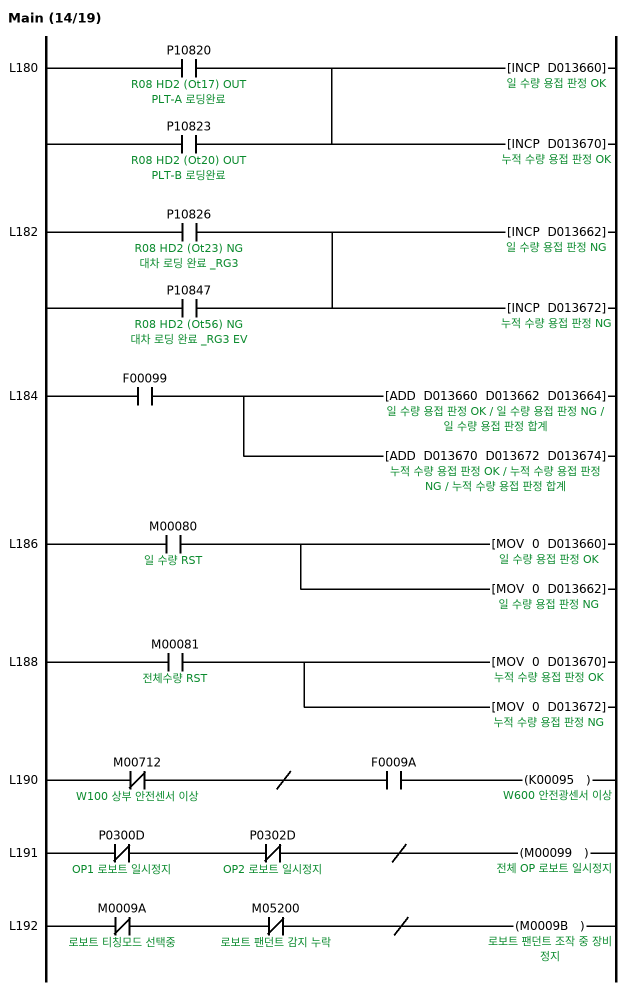
; L180
LOAD      P10820	// R08 HD2 (Ot17) OUT PLT-A 로딩완료
OR        P10823	// R08 HD2 (Ot20) OUT PLT-B 로딩완료
INCP      D013660	// 일 수량 용접 판정 OK
INCP      D013670	// 누적 수량 용접 판정 OK
; L182
LOAD      P10826	// R08 HD2 (Ot23) NG 대차 로딩 완료 _RG3
OR        P10847	// R08 HD2 (Ot56) NG 대차 로딩 완료 _RG3 EV
INCP      D013662	// 일 수량 용접 판정 NG
INCP      D013672	// 누적 수량 용접 판정 NG
; L184
LOAD      F00099
ADD       D013660 D013662 D013664	// 일 수량 용접 판정 OK / 일 수량 용접 판정 NG / 일 수량 용접 판정 합계
ADD       D013670 D013672 D013674	// 누적 수량 용접 판정 OK / 누적 수량 용접 판정 NG / 누적 수량 용접 판정 합계
; L186
LOAD      M00080	// 일 수량 RST
MOV       0 D013660	// 일 수량 용접 판정 OK
MOV       0 D013662	// 일 수량 용접 판정 NG
; L188
LOAD      M00081	// 전체수량 RST
MOV       0 D013670	// 누적 수량 용접 판정 OK
MOV       0 D013672	// 누적 수량 용접 판정 NG
; L190
LOAD NOT  M00712	// W100 상부 안전센서 이상
NOT
AND       F0009A
OUT       K00095	// W600 안전광센서 이상
; L191
LOAD NOT  P0300D	// OP1 로보트 일시정지
AND NOT   P0302D	// OP2 로보트 일시정지
NOT
OUT       M00099	// 전체 OP 로보트 일시정지
; L192
LOAD NOT  M0009A	// 로보트 티칭모드 선택중
AND NOT   M05200	// 로보트 팬던트 감지 누락
NOT
OUT       M0009B	// 로보트 팬던트 조작 중 장비 정지

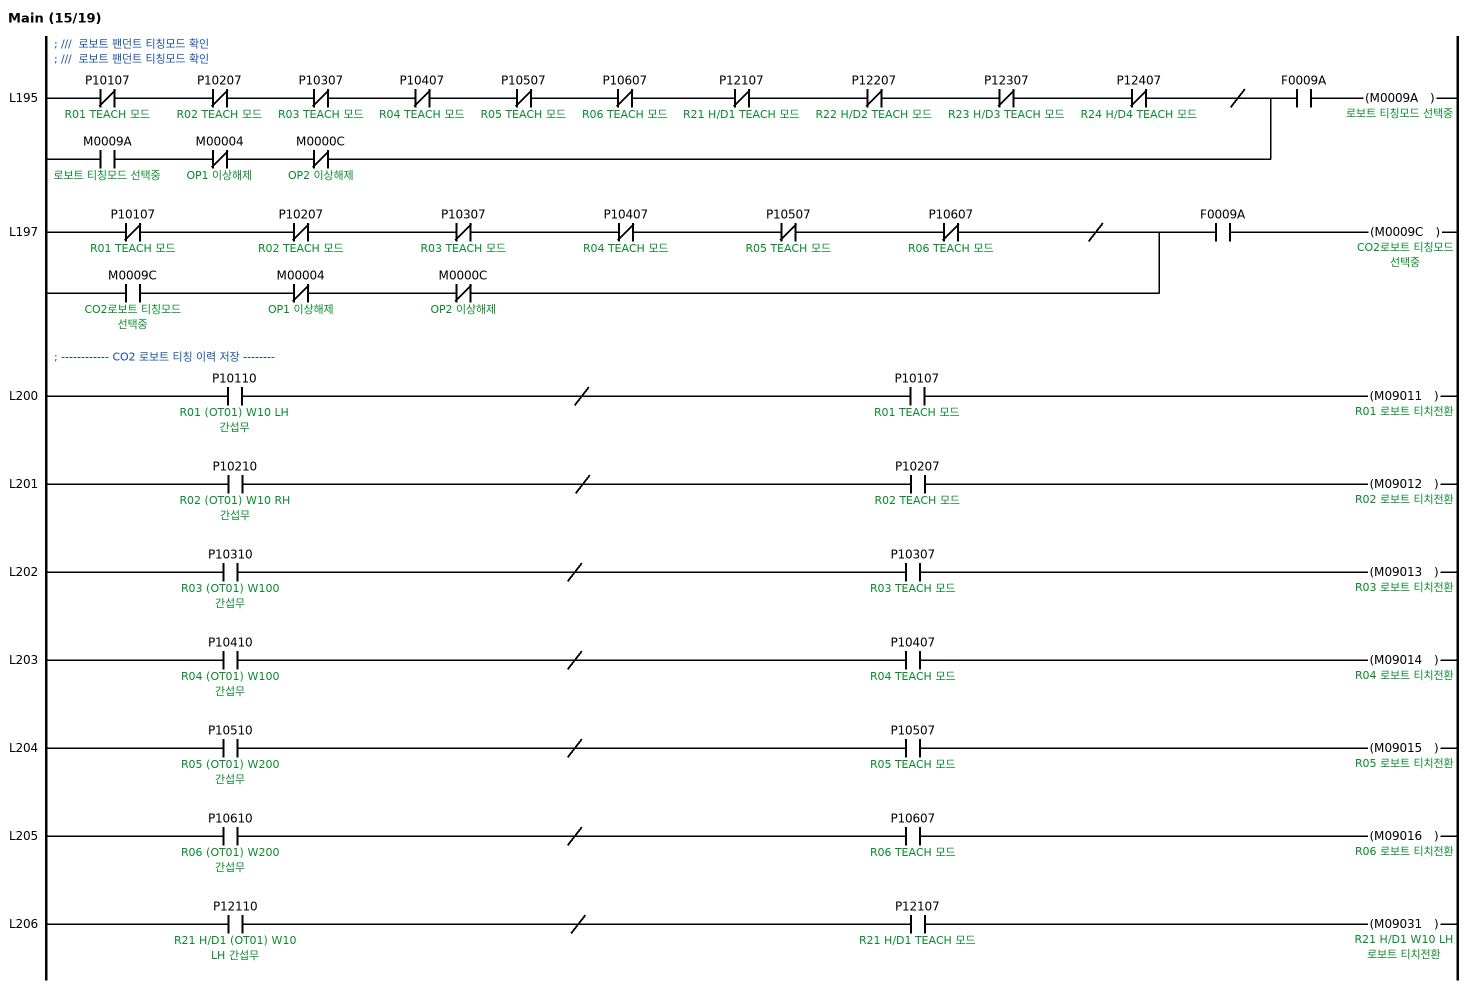
//    ///  로보트 팬던트 티칭모드 확인
//    ///  로보트 팬던트 티칭모드 확인
; L195
LOAD NOT  P10107	// R01 TEACH 모드
AND NOT   P10207	// R02 TEACH 모드
AND NOT   P10307	// R03 TEACH 모드
AND NOT   P10407	// R04 TEACH 모드
AND NOT   P10507	// R05 TEACH 모드
AND NOT   P10607	// R06 TEACH 모드
AND NOT   P12107	// R21 H/D1 TEACH 모드
AND NOT   P12207	// R22 H/D2 TEACH 모드
AND NOT   P12307	// R23 H/D3 TEACH 모드
AND NOT   P12407	// R24 H/D4 TEACH 모드
NOT
LOAD      M0009A	// 로보트 티칭모드 선택중
AND NOT   M00004	// OP1 이상해제
AND NOT   M0000C	// OP2 이상해제
OR LOAD
AND       F0009A
OUT       M0009A	// 로보트 티칭모드 선택중
; L197
LOAD NOT  P10107	// R01 TEACH 모드
AND NOT   P10207	// R02 TEACH 모드
AND NOT   P10307	// R03 TEACH 모드
AND NOT   P10407	// R04 TEACH 모드
AND NOT   P10507	// R05 TEACH 모드
AND NOT   P10607	// R06 TEACH 모드
NOT
LOAD      M0009C	// CO2로보트 티칭모드 선택중
AND NOT   M00004	// OP1 이상해제
AND NOT   M0000C	// OP2 이상해제
OR LOAD
AND       F0009A
OUT       M0009C	// CO2로보트 티칭모드 선택중
// ------------ CO2 로보트 티칭 이력 저장 --------
; L200
LOAD      P10110	// R01 (OT01) W10 LH 간섭무
NOT
AND       P10107	// R01 TEACH 모드
OUT       M09011	// R01 로보트 티치전환
; L201
LOAD      P10210	// R02 (OT01) W10 RH 간섭무
NOT
AND       P10207	// R02 TEACH 모드
OUT       M09012	// R02 로보트 티치전환
; L202
LOAD      P10310	// R03 (OT01) W100 간섭무
NOT
AND       P10307	// R03 TEACH 모드
OUT       M09013	// R03 로보트 티치전환
; L203
LOAD      P10410	// R04 (OT01) W100 간섭무
NOT
AND       P10407	// R04 TEACH 모드
OUT       M09014	// R04 로보트 티치전환
; L204
LOAD      P10510	// R05 (OT01) W200 간섭무
NOT
AND       P10507	// R05 TEACH 모드
OUT       M09015	// R05 로보트 티치전환
; L205
LOAD      P10610	// R06 (OT01) W200 간섭무
NOT
AND       P10607	// R06 TEACH 모드
OUT       M09016	// R06 로보트 티치전환
; L206
LOAD      P12110	// R21 H/D1 (OT01) W10 LH 간섭무
NOT
AND       P12107	// R21 H/D1 TEACH 모드
OUT       M09031	// R21 H/D1 W10 LH 로보트 티치전환

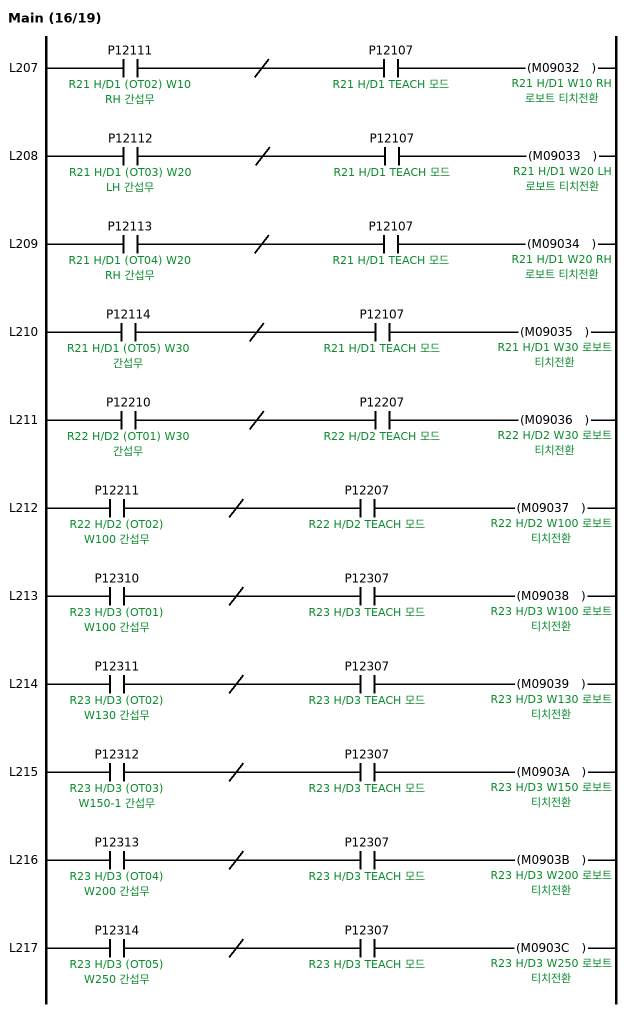
; L207
LOAD      P12111	// R21 H/D1 (OT02) W10 RH 간섭무
NOT
AND       P12107	// R21 H/D1 TEACH 모드
OUT       M09032	// R21 H/D1 W10 RH 로보트 티치전환
; L208
LOAD      P12112	// R21 H/D1 (OT03) W20 LH 간섭무
NOT
AND       P12107	// R21 H/D1 TEACH 모드
OUT       M09033	// R21 H/D1 W20 LH 로보트 티치전환
; L209
LOAD      P12113	// R21 H/D1 (OT04) W20 RH 간섭무
NOT
AND       P12107	// R21 H/D1 TEACH 모드
OUT       M09034	// R21 H/D1 W20 RH 로보트 티치전환
; L210
LOAD      P12114	// R21 H/D1 (OT05) W30 간섭무
NOT
AND       P12107	// R21 H/D1 TEACH 모드
OUT       M09035	// R21 H/D1 W30 로보트 티치전환
; L211
LOAD      P12210	// R22 H/D2 (OT01) W30 간섭무
NOT
AND       P12207	// R22 H/D2 TEACH 모드
OUT       M09036	// R22 H/D2 W30 로보트 티치전환
; L212
LOAD      P12211	// R22 H/D2 (OT02) W100 간섭무
NOT
AND       P12207	// R22 H/D2 TEACH 모드
OUT       M09037	// R22 H/D2 W100 로보트 티치전환
; L213
LOAD      P12310	// R23 H/D3 (OT01) W100 간섭무
NOT
AND       P12307	// R23 H/D3 TEACH 모드
OUT       M09038	// R23 H/D3 W100 로보트 티치전환
; L214
LOAD      P12311	// R23 H/D3 (OT02) W130 간섭무
NOT
AND       P12307	// R23 H/D3 TEACH 모드
OUT       M09039	// R23 H/D3 W130 로보트 티치전환
; L215
LOAD      P12312	// R23 H/D3 (OT03) W150-1 간섭무
NOT
AND       P12307	// R23 H/D3 TEACH 모드
OUT       M0903A	// R23 H/D3 W150 로보트 티치전환
; L216
LOAD      P12313	// R23 H/D3 (OT04) W200 간섭무
NOT
AND       P12307	// R23 H/D3 TEACH 모드
OUT       M0903B	// R23 H/D3 W200 로보트 티치전환
; L217
LOAD      P12314	// R23 H/D3 (OT05) W250 간섭무
NOT
AND       P12307	// R23 H/D3 TEACH 모드
OUT       M0903C	// R23 H/D3 W250 로보트 티치전환

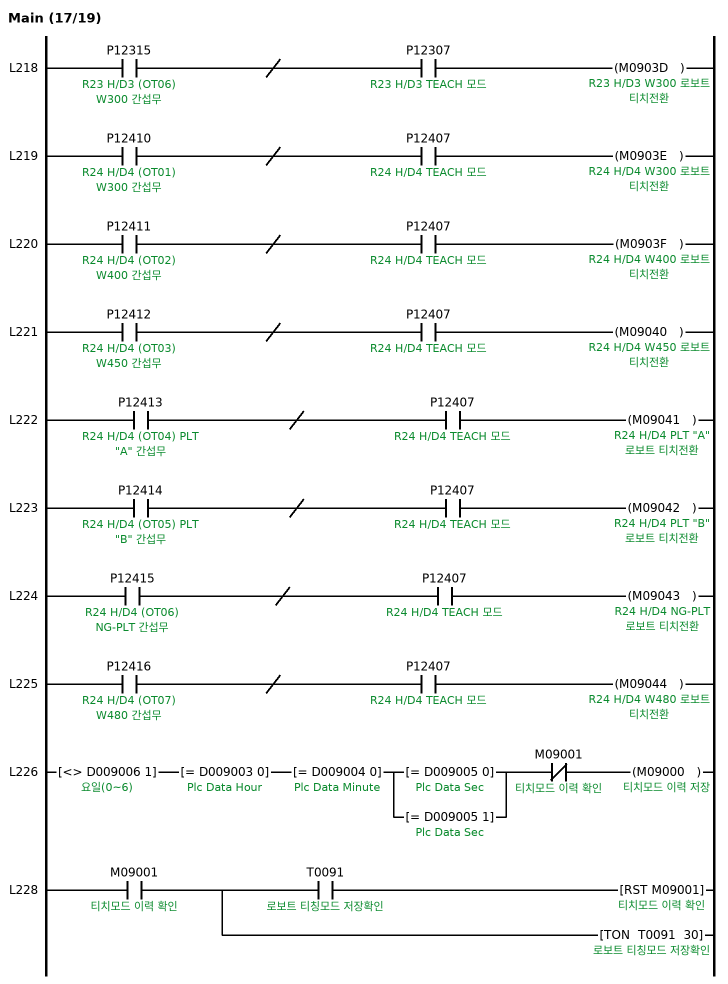
; L218
LOAD      P12315	// R23 H/D3 (OT06) W300 간섭무
NOT
AND       P12307	// R23 H/D3 TEACH 모드
OUT       M0903D	// R23 H/D3 W300 로보트 티치전환
; L219
LOAD      P12410	// R24 H/D4 (OT01) W300 간섭무
NOT
AND       P12407	// R24 H/D4 TEACH 모드
OUT       M0903E	// R24 H/D4 W300 로보트 티치전환
; L220
LOAD      P12411	// R24 H/D4 (OT02) W400 간섭무
NOT
AND       P12407	// R24 H/D4 TEACH 모드
OUT       M0903F	// R24 H/D4 W400 로보트 티치전환
; L221
LOAD      P12412	// R24 H/D4 (OT03) W450 간섭무
NOT
AND       P12407	// R24 H/D4 TEACH 모드
OUT       M09040	// R24 H/D4 W450 로보트 티치전환
; L222
LOAD      P12413	// R24 H/D4 (OT04) PLT "A" 간섭무
NOT
AND       P12407	// R24 H/D4 TEACH 모드
OUT       M09041	// R24 H/D4 PLT "A" 로보트 티치전환
; L223
LOAD      P12414	// R24 H/D4 (OT05) PLT "B" 간섭무
NOT
AND       P12407	// R24 H/D4 TEACH 모드
OUT       M09042	// R24 H/D4 PLT "B" 로보트 티치전환
; L224
LOAD      P12415	// R24 H/D4 (OT06) NG-PLT 간섭무
NOT
AND       P12407	// R24 H/D4 TEACH 모드
OUT       M09043	// R24 H/D4 NG-PLT 로보트 티치전환
; L225
LOAD      P12416	// R24 H/D4 (OT07) W480 간섭무
NOT
AND       P12407	// R24 H/D4 TEACH 모드
OUT       M09044	// R24 H/D4 W480 로보트 티치전환
; L226
LOAD<>    D009006 1	// 요일(0~6)
AND=      D009003 0	// Plc Data Hour
AND=      D009004 0	// Plc Data Minute
LOAD=     D009005 0	// Plc Data Sec
OR=       D009005 1	// Plc Data Sec
AND LOAD
AND NOT   M09001	// 티치모드 이력 확인
OUT       M09000	// 티치모드 이력 저장
; L228
LOAD      M09001	// 티치모드 이력 확인
MPUSH
AND       T0091	// 로보트 티칭모드 저장확인
RST       M09001	// 티치모드 이력 확인
MPOP
TON       T0091 30	// 로보트 티칭모드 저장확인

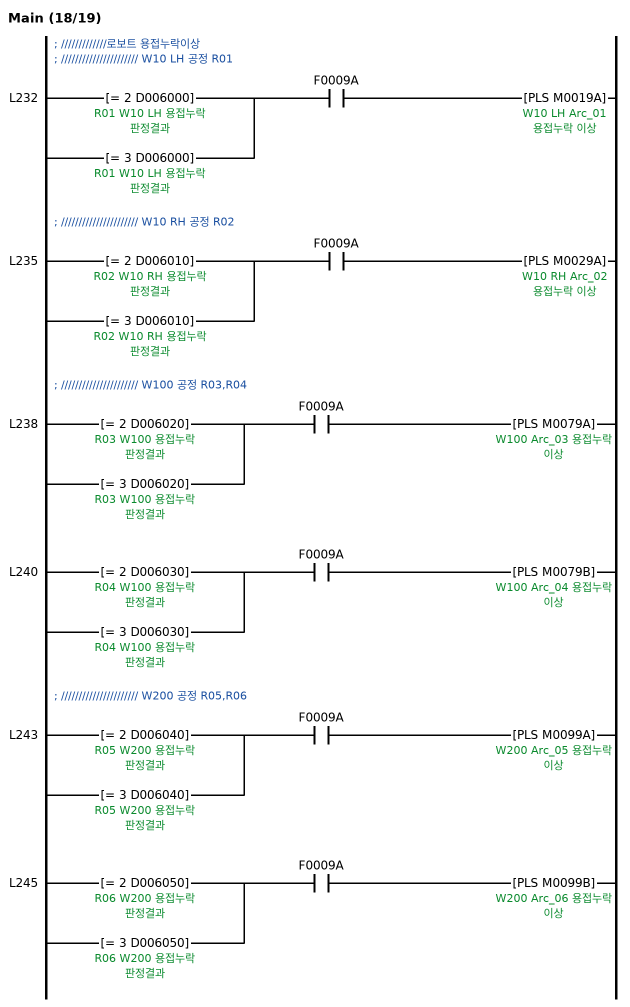
// /////////////로보트 용접누락이상
// ////////////////////// W10 LH 공정 R01
; L232
LOAD=     2 D006000	// R01 W10 LH 용접누락 판정결과
OR=       3 D006000	// R01 W10 LH 용접누락 판정결과
AND       F0009A
OUTP      M0019A	// W10 LH Arc_01 용접누락 이상
// ////////////////////// W10 RH 공정 R02
; L235
LOAD=     2 D006010	// R02 W10 RH 용접누락 판정결과
OR=       3 D006010	// R02 W10 RH 용접누락 판정결과
AND       F0009A
OUTP      M0029A	// W10 RH Arc_02 용접누락 이상
// ////////////////////// W100 공정 R03,R04
; L238
LOAD=     2 D006020	// R03 W100 용접누락 판정결과
OR=       3 D006020	// R03 W100 용접누락 판정결과
AND       F0009A
OUTP      M0079A	// W100 Arc_03 용접누락 이상
; L240
LOAD=     2 D006030	// R04 W100 용접누락 판정결과
OR=       3 D006030	// R04 W100 용접누락 판정결과
AND       F0009A
OUTP      M0079B	// W100 Arc_04 용접누락 이상
// ////////////////////// W200 공정 R05,R06
; L243
LOAD=     2 D006040	// R05 W200 용접누락 판정결과
OR=       3 D006040	// R05 W200 용접누락 판정결과
AND       F0009A
OUTP      M0099A	// W200 Arc_05 용접누락 이상
; L245
LOAD=     2 D006050	// R06 W200 용접누락 판정결과
OR=       3 D006050	// R06 W200 용접누락 판정결과
AND       F0009A
OUTP      M0099B	// W200 Arc_06 용접누락 이상

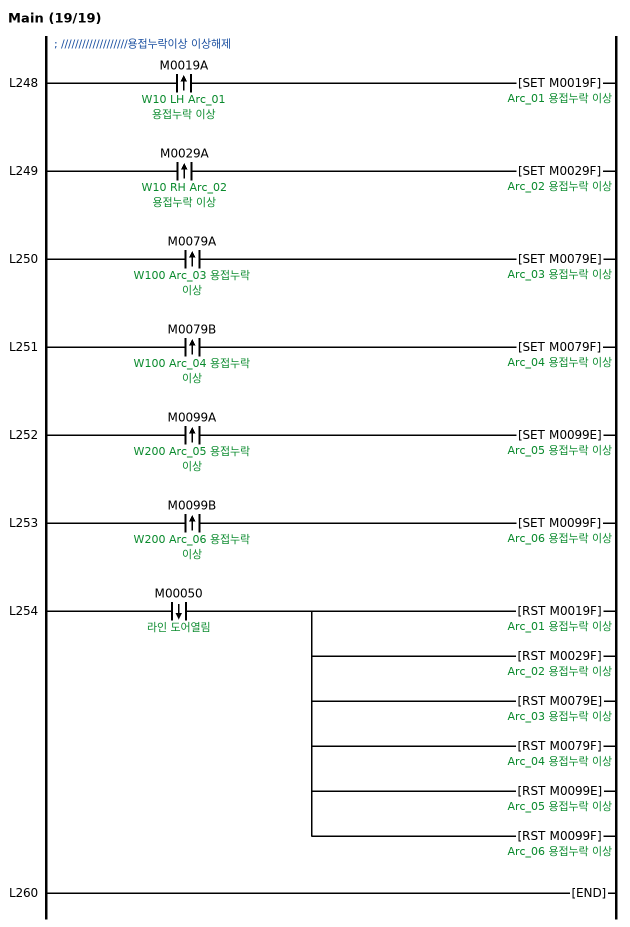
// ///////////////////용접누락이상 이상해제
; L248
LOADP     M0019A	// W10 LH Arc_01 용접누락 이상
SET       M0019F	// Arc_01 용접누락 이상
; L249
LOADP     M0029A	// W10 RH Arc_02 용접누락 이상
SET       M0029F	// Arc_02 용접누락 이상
; L250
LOADP     M0079A	// W100 Arc_03 용접누락 이상
SET       M0079E	// Arc_03 용접누락 이상
; L251
LOADP     M0079B	// W100 Arc_04 용접누락 이상
SET       M0079F	// Arc_04 용접누락 이상
; L252
LOADP     M0099A	// W200 Arc_05 용접누락 이상
SET       M0099E	// Arc_05 용접누락 이상
; L253
LOADP     M0099B	// W200 Arc_06 용접누락 이상
SET       M0099F	// Arc_06 용접누락 이상
; L254
LOADN     M00050	// 라인 도어열림
RST       M0019F	// Arc_01 용접누락 이상
RST       M0029F	// Arc_02 용접누락 이상
RST       M0079E	// Arc_03 용접누락 이상
RST       M0079F	// Arc_04 용접누락 이상
RST       M0099E	// Arc_05 용접누락 이상
RST       M0099F	// Arc_06 용접누락 이상
; L260
END

PROGRAM OP1 (task: 스캔 프로그램)

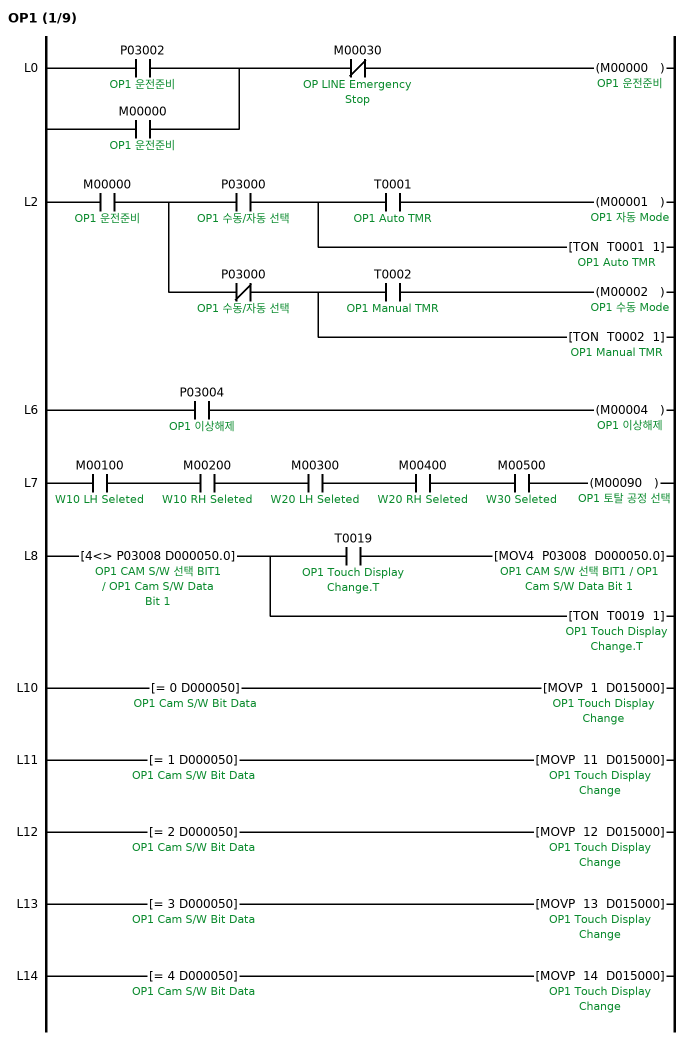
; L0
LOAD      P03002	// OP1 운전준비
OR        M00000	// OP1 운전준비
AND NOT   M00030	// OP LINE Emergency Stop
OUT       M00000	// OP1 운전준비
; L2
LOAD      M00000	// OP1 운전준비
MPUSH
AND       P03000	// OP1 수동/자동 선택
MPUSH
AND       T0001	// OP1 Auto TMR
OUT       M00001	// OP1 자동 Mode
MPOP
TON       T0001 1	// OP1 Auto TMR
MPOP
AND NOT   P03000	// OP1 수동/자동 선택
MPUSH
AND       T0002	// OP1 Manual TMR
OUT       M00002	// OP1 수동 Mode
MPOP
TON       T0002 1	// OP1 Manual TMR
; L6
LOAD      P03004	// OP1 이상해제
OUT       M00004	// OP1 이상해제
; L7
LOAD      M00100	// W10 LH Seleted
AND       M00200	// W10 RH Seleted
AND       M00300	// W20 LH Seleted
AND       M00400	// W20 RH Seleted
AND       M00500	// W30 Seleted
OUT       M00090	// OP1 토탈 공정 선택
; L8
LOAD4<>   P03008 D000050.0	// OP1 CAM S/W 선택 BIT1 / OP1 Cam S/W Data Bit 1
MPUSH
AND       T0019	// OP1 Touch Display Change.T
MOV4      P03008 D000050.0	// OP1 CAM S/W 선택 BIT1 / OP1 Cam S/W Data Bit 1
MPOP
TON       T0019 1	// OP1 Touch Display Change.T
; L10
LOAD=     0 D000050	// OP1 Cam S/W Bit Data
MOVP      1 D015000	// OP1 Touch Display Change
; L11
LOAD=     1 D000050	// OP1 Cam S/W Bit Data
MOVP      11 D015000	// OP1 Touch Display Change
; L12
LOAD=     2 D000050	// OP1 Cam S/W Bit Data
MOVP      12 D015000	// OP1 Touch Display Change
; L13
LOAD=     3 D000050	// OP1 Cam S/W Bit Data
MOVP      13 D015000	// OP1 Touch Display Change
; L14
LOAD=     4 D000050	// OP1 Cam S/W Bit Data
MOVP      14 D015000	// OP1 Touch Display Change

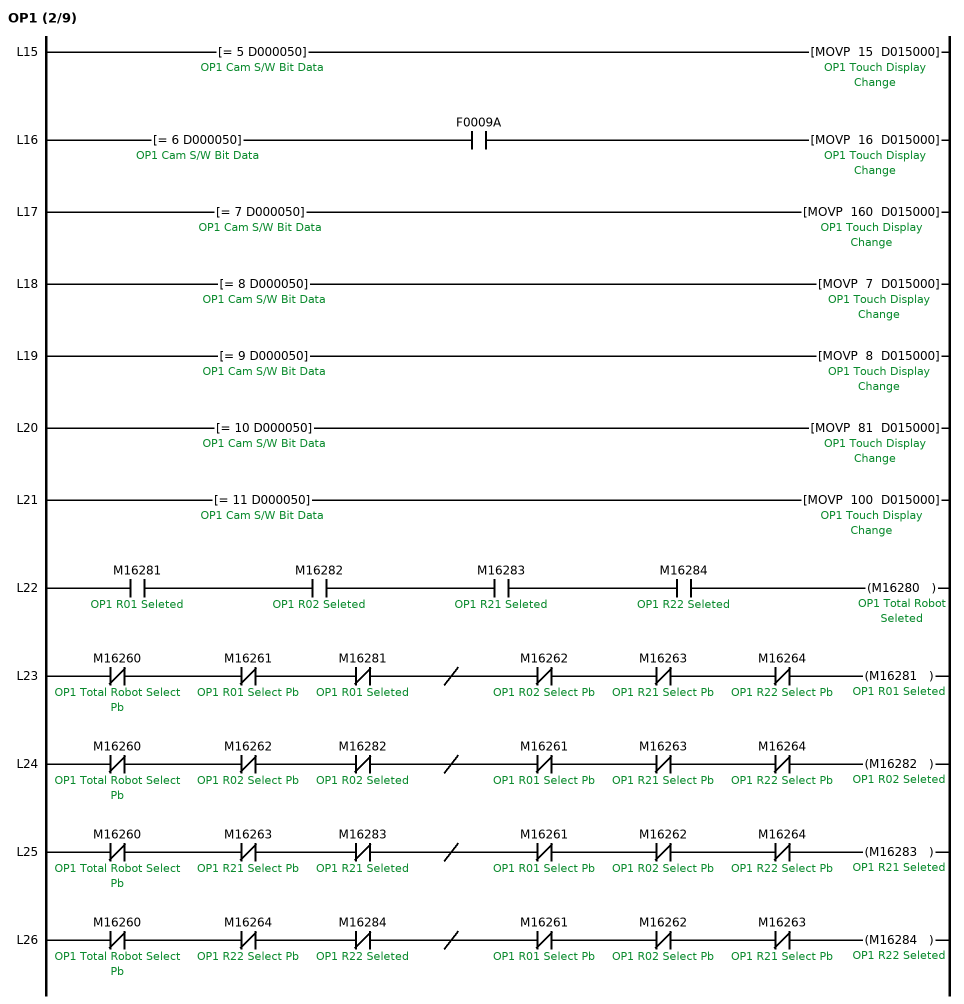
; L15
LOAD=     5 D000050	// OP1 Cam S/W Bit Data
MOVP      15 D015000	// OP1 Touch Display Change
; L16
LOAD=     6 D000050	// OP1 Cam S/W Bit Data
AND       F0009A
MOVP      16 D015000	// OP1 Touch Display Change
; L17
LOAD=     7 D000050	// OP1 Cam S/W Bit Data
MOVP      160 D015000	// OP1 Touch Display Change
; L18
LOAD=     8 D000050	// OP1 Cam S/W Bit Data
MOVP      7 D015000	// OP1 Touch Display Change
; L19
LOAD=     9 D000050	// OP1 Cam S/W Bit Data
MOVP      8 D015000	// OP1 Touch Display Change
; L20
LOAD=     10 D000050	// OP1 Cam S/W Bit Data
MOVP      81 D015000	// OP1 Touch Display Change
; L21
LOAD=     11 D000050	// OP1 Cam S/W Bit Data
MOVP      100 D015000	// OP1 Touch Display Change
; L22
LOAD      M16281	// OP1 R01 Seleted
AND       M16282	// OP1 R02 Seleted
AND       M16283	// OP1 R21 Seleted
AND       M16284	// OP1 R22 Seleted
OUT       M16280	// OP1 Total Robot Seleted
; L23
LOAD NOT  M16260	// OP1 Total Robot Select Pb
AND NOT   M16261	// OP1 R01 Select Pb
AND NOT   M16281	// OP1 R01 Seleted
NOT
AND NOT   M16262	// OP1 R02 Select Pb
AND NOT   M16263	// OP1 R21 Select Pb
AND NOT   M16264	// OP1 R22 Select Pb
OUT       M16281	// OP1 R01 Seleted
; L24
LOAD NOT  M16260	// OP1 Total Robot Select Pb
AND NOT   M16262	// OP1 R02 Select Pb
AND NOT   M16282	// OP1 R02 Seleted
NOT
AND NOT   M16261	// OP1 R01 Select Pb
AND NOT   M16263	// OP1 R21 Select Pb
AND NOT   M16264	// OP1 R22 Select Pb
OUT       M16282	// OP1 R02 Seleted
; L25
LOAD NOT  M16260	// OP1 Total Robot Select Pb
AND NOT   M16263	// OP1 R21 Select Pb
AND NOT   M16283	// OP1 R21 Seleted
NOT
AND NOT   M16261	// OP1 R01 Select Pb
AND NOT   M16262	// OP1 R02 Select Pb
AND NOT   M16264	// OP1 R22 Select Pb
OUT       M16283	// OP1 R21 Seleted
; L26
LOAD NOT  M16260	// OP1 Total Robot Select Pb
AND NOT   M16264	// OP1 R22 Select Pb
AND NOT   M16284	// OP1 R22 Seleted
NOT
AND NOT   M16261	// OP1 R01 Select Pb
AND NOT   M16262	// OP1 R02 Select Pb
AND NOT   M16263	// OP1 R21 Select Pb
OUT       M16284	// OP1 R22 Seleted

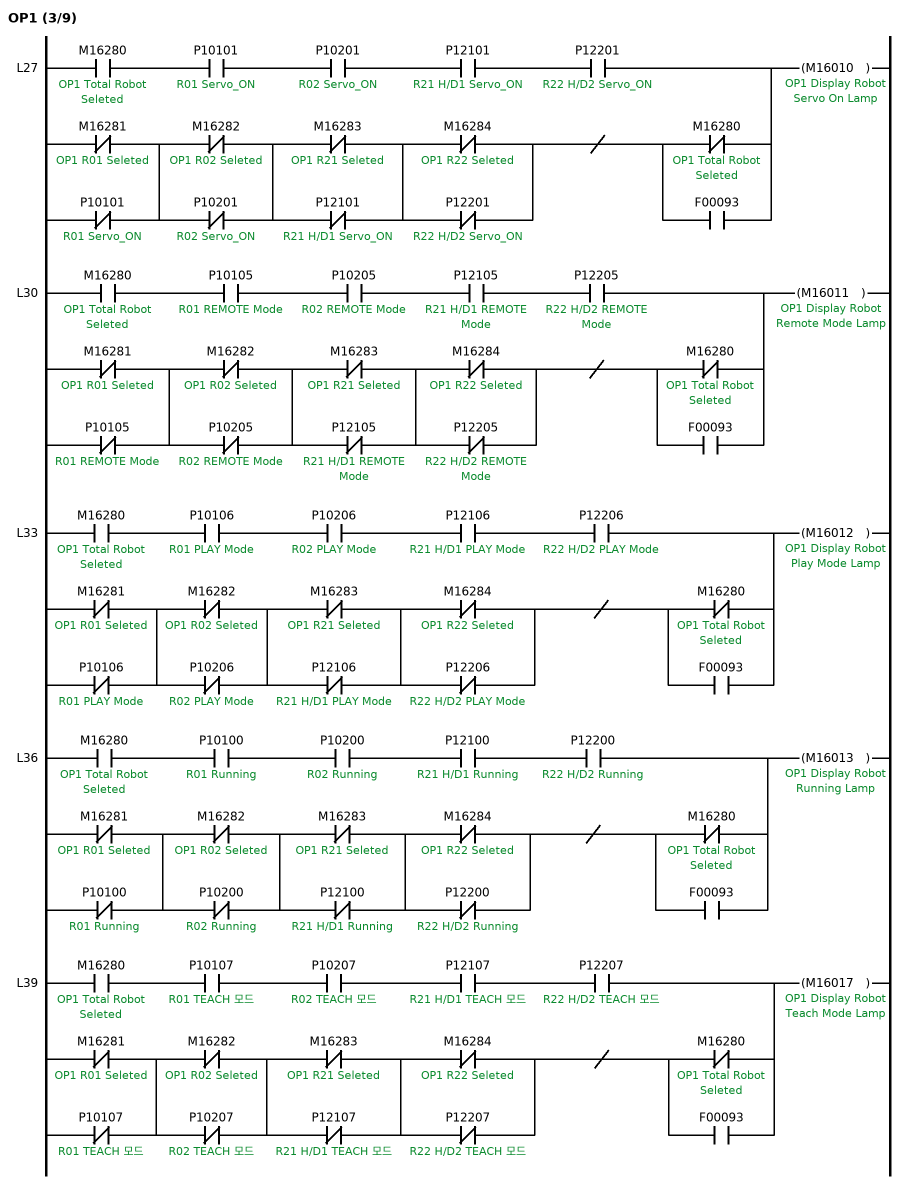
; L27
LOAD      M16280	// OP1 Total Robot Seleted
AND       P10101	// R01 Servo_ON
AND       P10201	// R02 Servo_ON
AND       P12101	// R21 H/D1 Servo_ON
AND       P12201	// R22 H/D2 Servo_ON
LOAD NOT  M16281	// OP1 R01 Seleted
OR NOT    P10101	// R01 Servo_ON
LOAD NOT  M16282	// OP1 R02 Seleted
OR NOT    P10201	// R02 Servo_ON
AND LOAD
LOAD NOT  M16283	// OP1 R21 Seleted
OR NOT    P12101	// R21 H/D1 Servo_ON
AND LOAD
LOAD NOT  M16284	// OP1 R22 Seleted
OR NOT    P12201	// R22 H/D2 Servo_ON
AND LOAD
NOT
LOAD NOT  M16280	// OP1 Total Robot Seleted
OR        F00093
AND LOAD
OR LOAD
OUT       M16010	// OP1 Display Robot Servo On Lamp
; L30
LOAD      M16280	// OP1 Total Robot Seleted
AND       P10105	// R01 REMOTE Mode
AND       P10205	// R02 REMOTE Mode
AND       P12105	// R21 H/D1 REMOTE Mode
AND       P12205	// R22 H/D2 REMOTE Mode
LOAD NOT  M16281	// OP1 R01 Seleted
OR NOT    P10105	// R01 REMOTE Mode
LOAD NOT  M16282	// OP1 R02 Seleted
OR NOT    P10205	// R02 REMOTE Mode
AND LOAD
LOAD NOT  M16283	// OP1 R21 Seleted
OR NOT    P12105	// R21 H/D1 REMOTE Mode
AND LOAD
LOAD NOT  M16284	// OP1 R22 Seleted
OR NOT    P12205	// R22 H/D2 REMOTE Mode
AND LOAD
NOT
LOAD NOT  M16280	// OP1 Total Robot Seleted
OR        F00093
AND LOAD
OR LOAD
OUT       M16011	// OP1 Display Robot Remote Mode Lamp
; L33
LOAD      M16280	// OP1 Total Robot Seleted
AND       P10106	// R01 PLAY Mode
AND       P10206	// R02 PLAY Mode
AND       P12106	// R21 H/D1 PLAY Mode
AND       P12206	// R22 H/D2 PLAY Mode
LOAD NOT  M16281	// OP1 R01 Seleted
OR NOT    P10106	// R01 PLAY Mode
LOAD NOT  M16282	// OP1 R02 Seleted
OR NOT    P10206	// R02 PLAY Mode
AND LOAD
LOAD NOT  M16283	// OP1 R21 Seleted
OR NOT    P12106	// R21 H/D1 PLAY Mode
AND LOAD
LOAD NOT  M16284	// OP1 R22 Seleted
OR NOT    P12206	// R22 H/D2 PLAY Mode
AND LOAD
NOT
LOAD NOT  M16280	// OP1 Total Robot Seleted
OR        F00093
AND LOAD
OR LOAD
OUT       M16012	// OP1 Display Robot Play Mode Lamp
; L36
LOAD      M16280	// OP1 Total Robot Seleted
AND       P10100	// R01 Running
AND       P10200	// R02 Running
AND       P12100	// R21 H/D1 Running
AND       P12200	// R22 H/D2 Running
LOAD NOT  M16281	// OP1 R01 Seleted
OR NOT    P10100	// R01 Running
LOAD NOT  M16282	// OP1 R02 Seleted
OR NOT    P10200	// R02 Running
AND LOAD
LOAD NOT  M16283	// OP1 R21 Seleted
OR NOT    P12100	// R21 H/D1 Running
AND LOAD
LOAD NOT  M16284	// OP1 R22 Seleted
OR NOT    P12200	// R22 H/D2 Running
AND LOAD
NOT
LOAD NOT  M16280	// OP1 Total Robot Seleted
OR        F00093
AND LOAD
OR LOAD
OUT       M16013	// OP1 Display Robot Running Lamp
; L39
LOAD      M16280	// OP1 Total Robot Seleted
AND       P10107	// R01 TEACH 모드
AND       P10207	// R02 TEACH 모드
AND       P12107	// R21 H/D1 TEACH 모드
AND       P12207	// R22 H/D2 TEACH 모드
LOAD NOT  M16281	// OP1 R01 Seleted
OR NOT    P10107	// R01 TEACH 모드
LOAD NOT  M16282	// OP1 R02 Seleted
OR NOT    P10207	// R02 TEACH 모드
AND LOAD
LOAD NOT  M16283	// OP1 R21 Seleted
OR NOT    P12107	// R21 H/D1 TEACH 모드
AND LOAD
LOAD NOT  M16284	// OP1 R22 Seleted
OR NOT    P12207	// R22 H/D2 TEACH 모드
AND LOAD
NOT
LOAD NOT  M16280	// OP1 Total Robot Seleted
OR        F00093
AND LOAD
OR LOAD
OUT       M16017	// OP1 Display Robot Teach Mode Lamp

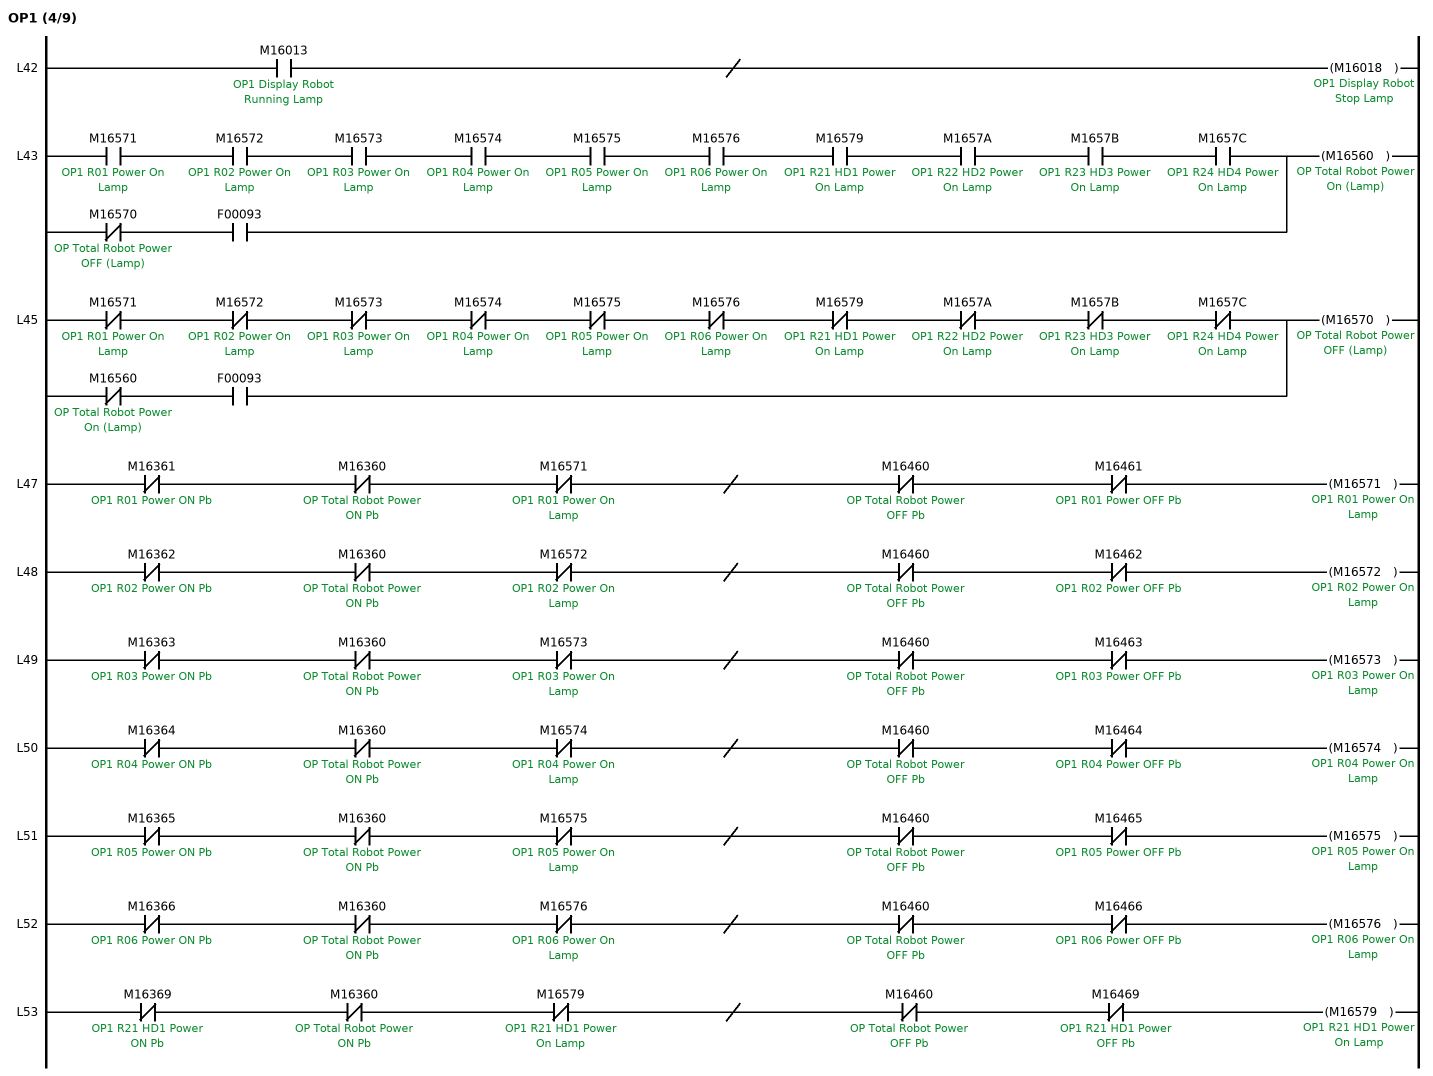
; L42
LOAD      M16013	// OP1 Display Robot Running Lamp
NOT
OUT       M16018	// OP1 Display Robot Stop Lamp
; L43
LOAD      M16571	// OP1 R01 Power On Lamp
AND       M16572	// OP1 R02 Power On Lamp
AND       M16573	// OP1 R03 Power On Lamp
AND       M16574	// OP1 R04 Power On Lamp
AND       M16575	// OP1 R05 Power On Lamp
AND       M16576	// OP1 R06 Power On Lamp
AND       M16579	// OP1 R21 HD1 Power On Lamp
AND       M1657A	// OP1 R22 HD2 Power On Lamp
AND       M1657B	// OP1 R23 HD3 Power On Lamp
AND       M1657C	// OP1 R24 HD4 Power On Lamp
LOAD NOT  M16570	// OP Total Robot Power OFF (Lamp)
AND       F00093
OR LOAD
OUT       M16560	// OP Total Robot Power On (Lamp)
; L45
LOAD NOT  M16571	// OP1 R01 Power On Lamp
AND NOT   M16572	// OP1 R02 Power On Lamp
AND NOT   M16573	// OP1 R03 Power On Lamp
AND NOT   M16574	// OP1 R04 Power On Lamp
AND NOT   M16575	// OP1 R05 Power On Lamp
AND NOT   M16576	// OP1 R06 Power On Lamp
AND NOT   M16579	// OP1 R21 HD1 Power On Lamp
AND NOT   M1657A	// OP1 R22 HD2 Power On Lamp
AND NOT   M1657B	// OP1 R23 HD3 Power On Lamp
AND NOT   M1657C	// OP1 R24 HD4 Power On Lamp
LOAD NOT  M16560	// OP Total Robot Power On (Lamp)
AND       F00093
OR LOAD
OUT       M16570	// OP Total Robot Power OFF (Lamp)
; L47
LOAD NOT  M16361	// OP1 R01 Power ON Pb
AND NOT   M16360	// OP Total Robot Power ON Pb
AND NOT   M16571	// OP1 R01 Power On Lamp
NOT
AND NOT   M16460	// OP Total Robot Power OFF Pb
AND NOT   M16461	// OP1 R01 Power OFF Pb
OUT       M16571	// OP1 R01 Power On Lamp
; L48
LOAD NOT  M16362	// OP1 R02 Power ON Pb
AND NOT   M16360	// OP Total Robot Power ON Pb
AND NOT   M16572	// OP1 R02 Power On Lamp
NOT
AND NOT   M16460	// OP Total Robot Power OFF Pb
AND NOT   M16462	// OP1 R02 Power OFF Pb
OUT       M16572	// OP1 R02 Power On Lamp
; L49
LOAD NOT  M16363	// OP1 R03 Power ON Pb
AND NOT   M16360	// OP Total Robot Power ON Pb
AND NOT   M16573	// OP1 R03 Power On Lamp
NOT
AND NOT   M16460	// OP Total Robot Power OFF Pb
AND NOT   M16463	// OP1 R03 Power OFF Pb
OUT       M16573	// OP1 R03 Power On Lamp
; L50
LOAD NOT  M16364	// OP1 R04 Power ON Pb
AND NOT   M16360	// OP Total Robot Power ON Pb
AND NOT   M16574	// OP1 R04 Power On Lamp
NOT
AND NOT   M16460	// OP Total Robot Power OFF Pb
AND NOT   M16464	// OP1 R04 Power OFF Pb
OUT       M16574	// OP1 R04 Power On Lamp
; L51
LOAD NOT  M16365	// OP1 R05 Power ON Pb
AND NOT   M16360	// OP Total Robot Power ON Pb
AND NOT   M16575	// OP1 R05 Power On Lamp
NOT
AND NOT   M16460	// OP Total Robot Power OFF Pb
AND NOT   M16465	// OP1 R05 Power OFF Pb
OUT       M16575	// OP1 R05 Power On Lamp
; L52
LOAD NOT  M16366	// OP1 R06 Power ON Pb
AND NOT   M16360	// OP Total Robot Power ON Pb
AND NOT   M16576	// OP1 R06 Power On Lamp
NOT
AND NOT   M16460	// OP Total Robot Power OFF Pb
AND NOT   M16466	// OP1 R06 Power OFF Pb
OUT       M16576	// OP1 R06 Power On Lamp
; L53
LOAD NOT  M16369	// OP1 R21 HD1 Power ON Pb
AND NOT   M16360	// OP Total Robot Power ON Pb
AND NOT   M16579	// OP1 R21 HD1 Power On Lamp
NOT
AND NOT   M16460	// OP Total Robot Power OFF Pb
AND NOT   M16469	// OP1 R21 HD1 Power OFF Pb
OUT       M16579	// OP1 R21 HD1 Power On Lamp

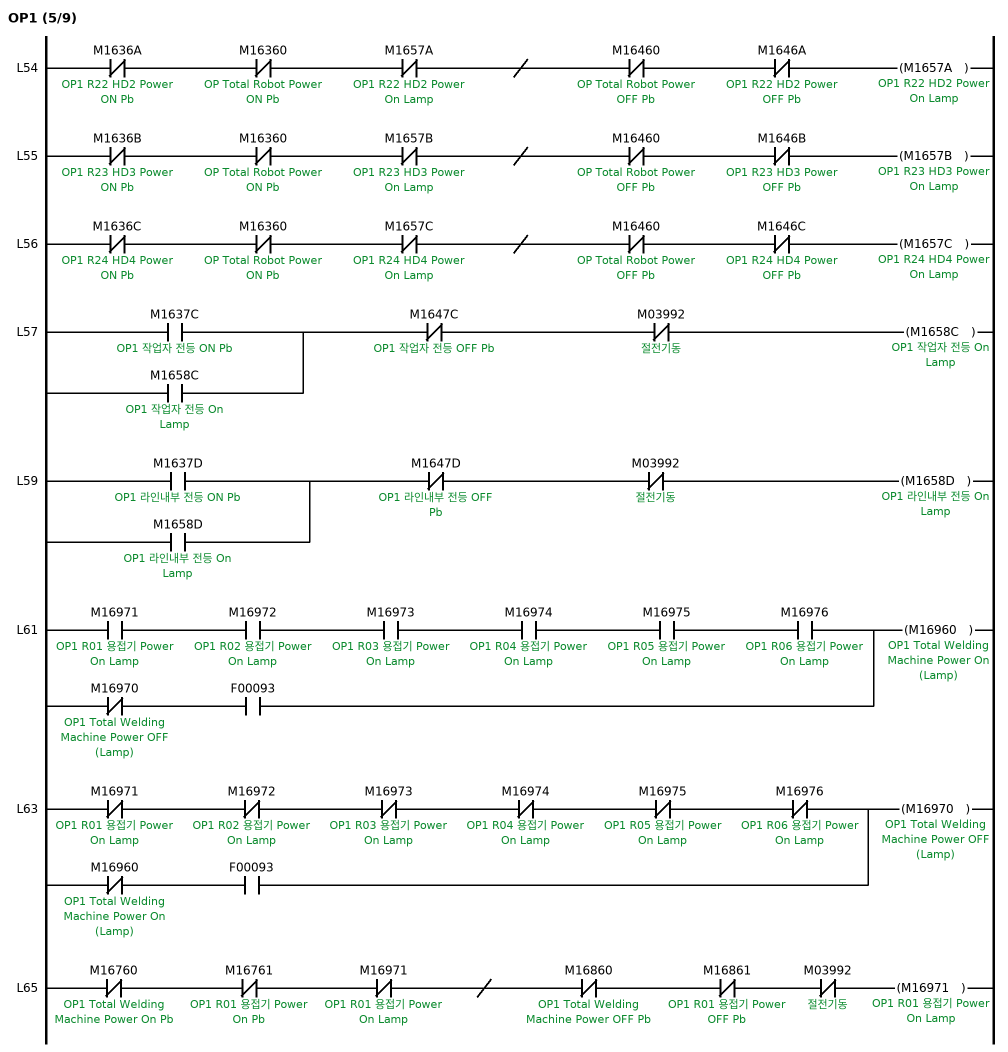
; L54
LOAD NOT  M1636A	// OP1 R22 HD2 Power ON Pb
AND NOT   M16360	// OP Total Robot Power ON Pb
AND NOT   M1657A	// OP1 R22 HD2 Power On Lamp
NOT
AND NOT   M16460	// OP Total Robot Power OFF Pb
AND NOT   M1646A	// OP1 R22 HD2 Power OFF Pb
OUT       M1657A	// OP1 R22 HD2 Power On Lamp
; L55
LOAD NOT  M1636B	// OP1 R23 HD3 Power ON Pb
AND NOT   M16360	// OP Total Robot Power ON Pb
AND NOT   M1657B	// OP1 R23 HD3 Power On Lamp
NOT
AND NOT   M16460	// OP Total Robot Power OFF Pb
AND NOT   M1646B	// OP1 R23 HD3 Power OFF Pb
OUT       M1657B	// OP1 R23 HD3 Power On Lamp
; L56
LOAD NOT  M1636C	// OP1 R24 HD4 Power ON Pb
AND NOT   M16360	// OP Total Robot Power ON Pb
AND NOT   M1657C	// OP1 R24 HD4 Power On Lamp
NOT
AND NOT   M16460	// OP Total Robot Power OFF Pb
AND NOT   M1646C	// OP1 R24 HD4 Power OFF Pb
OUT       M1657C	// OP1 R24 HD4 Power On Lamp
; L57
LOAD      M1637C	// OP1 작업자 전등 ON Pb
OR        M1658C	// OP1 작업자 전등 On Lamp
AND NOT   M1647C	// OP1 작업자 전등 OFF Pb
AND NOT   M03992	// 절전기동
OUT       M1658C	// OP1 작업자 전등 On Lamp
; L59
LOAD      M1637D	// OP1 라인내부 전등 ON Pb
OR        M1658D	// OP1 라인내부 전등 On Lamp
AND NOT   M1647D	// OP1 라인내부 전등 OFF Pb
AND NOT   M03992	// 절전기동
OUT       M1658D	// OP1 라인내부 전등 On Lamp
; L61
LOAD      M16971	// OP1 R01 용접기 Power On Lamp
AND       M16972	// OP1 R02 용접기 Power On Lamp
AND       M16973	// OP1 R03 용접기 Power On Lamp
AND       M16974	// OP1 R04 용접기 Power On Lamp
AND       M16975	// OP1 R05 용접기 Power On Lamp
AND       M16976	// OP1 R06 용접기 Power On Lamp
LOAD NOT  M16970	// OP1 Total Welding Machine Power OFF (Lamp)
AND       F00093
OR LOAD
OUT       M16960	// OP1 Total Welding Machine Power On (Lamp)
; L63
LOAD NOT  M16971	// OP1 R01 용접기 Power On Lamp
AND NOT   M16972	// OP1 R02 용접기 Power On Lamp
AND NOT   M16973	// OP1 R03 용접기 Power On Lamp
AND NOT   M16974	// OP1 R04 용접기 Power On Lamp
AND NOT   M16975	// OP1 R05 용접기 Power On Lamp
AND NOT   M16976	// OP1 R06 용접기 Power On Lamp
LOAD NOT  M16960	// OP1 Total Welding Machine Power On (Lamp)
AND       F00093
OR LOAD
OUT       M16970	// OP1 Total Welding Machine Power OFF (Lamp)
; L65
LOAD NOT  M16760	// OP1 Total Welding Machine Power On Pb
AND NOT   M16761	// OP1 R01 용접기 Power On Pb
AND NOT   M16971	// OP1 R01 용접기 Power On Lamp
NOT
AND NOT   M16860	// OP1 Total Welding Machine Power OFF Pb
AND NOT   M16861	// OP1 R01 용접기 Power OFF Pb
AND NOT   M03992	// 절전기동
OUT       M16971	// OP1 R01 용접기 Power On Lamp

